KUKA KRL program: MyProgram_184().src

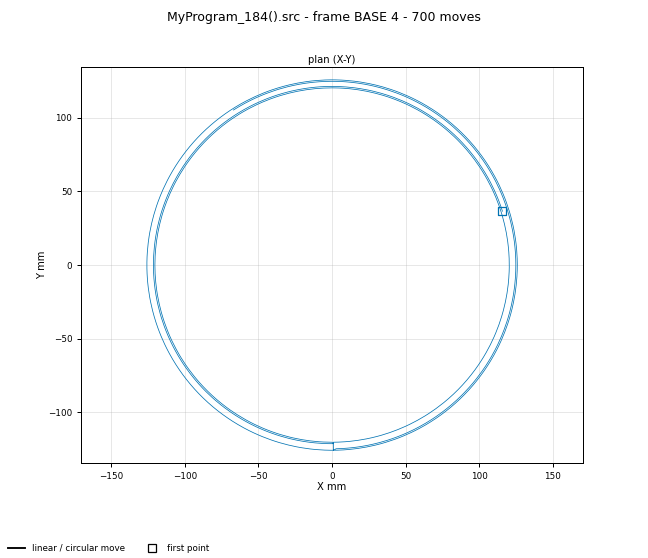
[picture p0: tool path of MyProgram_184().src in frame BASE 4, 700 of 700 moves have a stored position in this frame; points joined in program order, loops and branches not executed]
&ACCESS RVP
&REL 1
&PARAM TEMPLATE = C:\KRC\Roboter\Template\vorgabe
&PARAM EDITMASK = *
DEF MyProgram_184()
; ---- Setting reference (Base) ----
$BASE = BASE_DATA[4]

; --------------------------
; ---- Setting tool (TCP) ----
$TOOL = TOOL_DATA[3]
; --------------------------

$VEL.CP = VEL_APROX_PRINT
Startdeposition()
$VEL.CP = VEL_PRINT
LIN {X 115.7035,Y 36.5639,Z 134,A 13.9584,B 24.9464,C -1.6919,E1 25.152,E2 432.1213} C_DIS
LIN {X 114.6325,Y 39.7928,Z 134,A 15.5805,B 24.946,C -1.6976,E1 25.1505,E2 430.4949} C_DIS
LIN {X 113.3894,Y 43.2135,Z 134,A 17.3486,B 24.9455,C -1.7052,E1 25.1488,E2 428.7188} C_DIS
LIN {X 111.8645,Y 47.0156,Z 134,A 19.1684,B 24.9455,C -1.7052,E1 25.1469,E2 426.909} C_DIS
LIN {X 110.1148,Y 50.9782,Z 134,A 22.0831,B 24.9423,C -1.7548,E1 25.1434,E2 423.8932} C_DIS
LIN {X 107.5001,Y 56.2833,Z 134,A 23.673,B 24.9457,C -1.7024,E1 25.1415,E2 422.4351} C_DIS
LIN {X 105.7719,Y 59.4711,Z 134,A 25.7493,B 24.9442,C -1.7252,E1 25.1387,E2 420.3159} C_DIS
LIN {X 103.9941,Y 62.5285,Z 134,A 27.4667,B 24.9438,C -1.7321,E1 25.1362,E2 418.5912} C_DIS
LIN {X 101.7057,Y 66.1851,Z 134,A 30.2427,B 24.941,C -1.7744,E1 25.1319,E2 415.7292} C_DIS
LIN {X 98.373,Y 71.0443,Z 134,A 32.0344,B 24.9438,C -1.7322,E1 25.1292,E2 414.0459} C_DIS
LIN {X 96.2814,Y 73.854,Z 134,A 33.8484,B 24.943,C -1.7442,E1 25.1261,E2 412.2122} C_DIS
LIN {X 93.5282,Y 77.311,Z 134,A 35.9383,B 24.9426,C -1.7494,E1 25.1224,E2 410.1198} C_DIS
LIN {X 91.0407,Y 80.2255,Z 134,A 37.6345,B 24.9427,C -1.748,E1 25.1193,E2 408.4343} C_DIS
LIN {X 88.4927,Y 83.028,Z 134,A 39.4915,B 24.9422,C -1.7555,E1 25.1157,E2 406.568} C_DIS
LIN {X 86.0476,Y 85.5588,Z 134,A 41.1558,B 24.942,C -1.7592,E1 25.1125,E2 404.9019} C_DIS
LIN {X 82.9492,Y 88.5666,Z 134,A 43.0973,B 24.942,C -1.7588,E1 25.1086,E2 402.9694} C_DIS
LIN {X 80.4891,Y 90.8076,Z 134,A 44.7795,B 24.9415,C -1.7674,E1 25.1051,E2 401.2736} C_DIS
LIN {X 77.0787,Y 93.7202,Z 134,A 46.7789,B 24.9415,C -1.7658,E1 25.1008,E2 399.2857} C_DIS
LIN {X 73.9909,Y 96.1767,Z 134,A 48.7646,B 24.9409,C -1.7752,E1 25.0964,E2 397.2851} C_DIS
LIN {X 70.2941,Y 98.9108,Z 134,A 50.8899,B 24.9409,C -1.7768,E1 25.0916,E2 395.1636} C_DIS
LIN {X 65.6768,Y 102.035,Z 134,A 53.1943,B 24.9416,C -1.7653,E1 25.0864,E2 392.894} C_DIS
LIN {X 60.798,Y 105.0148,Z 134,A 56.0562,B 24.9408,C -1.7772,E1 25.0795,E2 390.0129} C_DIS
LIN {X 57.6858,Y 106.7564,Z 134,A 57.8367,B 24.9403,C -1.7842,E1 25.0751,E2 388.221} C_DIS
LIN {X 54.4905,Y 108.4215,Z 134,A 59.4404,B 24.9405,C -1.7818,E1 25.0711,E2 386.6275} C_DIS
LIN {X 52.1195,Y 109.5794,Z 134,A 61.0144,B 24.9393,C -1.7991,E1 25.0671,E2 385.0168} C_DIS
LIN {X 47.8558,Y 111.5078,Z 134,A 62.9444,B 24.9401,C -1.7882,E1 25.0622,E2 383.1172} C_DIS
LIN {X 41.891,Y 113.8847,Z 134,A 65.9124,B 24.9401,C -1.7882,E1 25.0545,E2 380.1559} C_DIS
LIN {X 37.7378,Y 115.3271,Z 134,A 68.2029,B 24.9393,C -1.8001,E1 25.0484,E2 377.8415} C_DIS
LIN {X 33.3869,Y 116.6617,Z 134,A 70.1325,B 24.9399,C -1.7913,E1 25.0433,E2 375.936} C_DIS
LIN {X 30.1024,Y 117.5501,Z 134,A 71.634,B 24.9401,C -1.7874,E1 25.0393,E2 374.4461} C_DIS
LIN {X 27.9003,Y 118.0931,Z 134,A 72.7821,B 24.9398,C -1.7917,E1 25.0361,E2 373.2896} C_DIS
LIN {X 24.6816,Y 118.8073,Z 134,A 74.2624,B 24.94,C -1.7889,E1 25.0321,E2 371.8179} C_DIS
LIN {X 21.5993,Y 119.4054,Z 134,A 75.6288,B 24.9403,C -1.7841,E1 25.0284,E2 370.4644} C_DIS
LIN {X 19.0604,Y 119.8377,Z 134,A 77.1116,B 24.9395,C -1.7969,E1 25.0242,E2 368.9527} C_DIS
LIN {X 15.3542,Y 120.3684,Z 134,A 79.0415,B 24.9389,C -1.8049,E1 25.0188,E2 367.0054} C_DIS
LIN {X 9.5046,Y 120.9722,Z 134,A 81.5766,B 24.9397,C -1.7939,E1 25.0119,E2 364.4979} C_DIS
LIN {X 4.175,Y 121.2715,Z 134,A 84.0832,B 24.9397,C -1.7932,E1 25.0049,E2 361.9938} C_DIS
LIN {X -3.3352,Y 121.2974,Z 134,A 87.3752,B 24.9406,C -1.7807,E1 24.9958,E2 358.7316} C_DIS
LIN {X -8.0647,Y 121.0756,Z 134,A 89.9951,B 24.9394,C -1.7975,E1 24.9884,E2 356.0711} C_DIS
LIN {X -10.9283,Y 120.8515,Z 134,A 91.8989,B 24.9378,C -1.8221,E1 24.9829,E2 354.1081} C_DIS
LIN {X -15.3011,Y 120.3754,Z 134,A 93.3926,B 24.9397,C -1.794,E1 24.9789,E2 352.68} C_DIS
LIN {X -18.4282,Y 119.9356,Z 134,A 94.8364,B 24.9399,C -1.7909,E1 24.975,E2 351.2425} C_DIS
LIN {X -23.1856,Y 119.108,Z 134,A 97.1985,B 24.9398,C -1.7928,E1 24.9685,E2 348.8734} C_DIS
LIN {X -27.8258,Y 118.1111,Z 134,A 99.3651,B 24.9401,C -1.7874,E1 24.9626,E2 346.7169} C_DIS
LIN {X -30.2861,Y 117.5034,Z 134,A 100.7404,B 24.9397,C -1.7943,E1 24.9588,E2 345.3231} C_DIS
LIN {X -33.7688,Y 116.5499,Z 134,A 102.3978,B 24.9399,C -1.7903,E1 24.9544,E2 343.6725} C_DIS
LIN {X -36.9708,Y 115.5736,Z 134,A 103.902,B 24.9403,C -1.785,E1 24.9504,E2 342.1783} C_DIS
LIN {X -40.2534,Y 114.4728,Z 134,A 105.5084,B 24.9405,C -1.7817,E1 24.9462,E2 340.5768} C_DIS
LIN {X -44.5725,Y 112.8618,Z 134,A 107.6515,B 24.9408,C -1.7772,E1 24.9406,E2 338.4398} C_DIS
LIN {X -47.2777,Y 111.7551,Z 134,A 109.0429,B 24.9408,C -1.7758,E1 24.937,E2 337.0487} C_DIS
LIN {X -49.6424,Y 110.7236,Z 134,A 110.3052,B 24.9408,C -1.7759,E1 24.9338,E2 335.783} C_DIS
LIN {X -52.8834,Y 109.2145,Z 134,A 111.9711,B 24.9411,C -1.7722,E1 24.9296,E2 334.1216} C_DIS
LIN {X -55.7632,Y 107.7732,Z 134,A 113.7041,B 24.9407,C -1.7792,E1 24.9252,E2 332.3674} C_DIS
LIN {X -59.7868,Y 105.5944,Z 134,A 115.8609,B 24.9409,C -1.7752,E1 24.9199,E2 330.2138} C_DIS
LIN {X -63.7405,Y 103.2558,Z 134,A 117.8702,B 24.9417,C -1.7641,E1 24.9152,E2 328.2248} C_DIS
LIN {X -66.727,Y 101.3509,Z 134,A 119.6469,B 24.9416,C -1.7655,E1 24.911,E2 326.4391} C_DIS
LIN {X -70.2515,Y 98.9412,Z 134,A 121.7402,B 24.9416,C -1.7648,E1 24.9062,E2 324.3403} C_DIS
LIN {X -73.8247,Y 96.3038,Z 134,A 123.7505,B 24.9422,C -1.7565,E1 24.9017,E2 322.3425} C_DIS
LIN {X -76.7002,Y 94.0297,Z 134,A 125.5201,B 24.9423,C -1.7544,E1 24.8979,E2 320.5713} C_DIS
LIN {X -79.9876,Y 91.25,Z 134,A 127.6022,B 24.9425,C -1.7519,E1 24.8935,E2 318.487} C_DIS
LIN {X -83.0686,Y 88.4544,Z 134,A 129.5856,B 24.9427,C -1.7481,E1 24.8894,E2 316.5046} C_DIS
LIN {X -85.974,Y 85.6329,Z 134,A 131.4349,B 24.9432,C -1.7407,E1 24.8858,E2 314.6652} C_DIS
LIN {X -88.6608,Y 82.8481,Z 134,A 133.3372,B 24.9433,C -1.7394,E1 24.8821,E2 312.7578} C_DIS
LIN {X -91.6123,Y 79.5724,Z 134,A 135.3816,B 24.9438,C -1.7323,E1 24.8783,E2 310.7208} C_DIS
LIN {X -94.2611,Y 76.4161,Z 134,A 137.3068,B 24.9442,C -1.7263,E1 24.8749,E2 308.8012} C_DIS
LIN {X -96.6023,Y 73.4344,Z 134,A 139.2073,B 24.9442,C -1.7263,E1 24.8716,E2 306.8918} C_DIS
LIN {X -99.1829,Y 69.9088,Z 134,A 141.2347,B 24.9446,C -1.719,E1 24.8684,E2 304.8718} C_DIS
LIN {X -101.1758,Y 66.993,Z 134,A 143.5278,B 24.9432,C -1.7416,E1 24.8647,E2 302.5132} C_DIS
LIN {X -103.799,Y 62.8512,Z 134,A 144.9179,B 24.9462,C -1.6946,E1 24.8629,E2 301.2282} C_DIS
LIN {X -105.1935,Y 60.4893,Z 134,A 147.3202,B 24.9433,C -1.7391,E1 24.8594,E2 298.7073} C_DIS
LIN {X -107.8811,Y 55.552,Z 134,A 149.3952,B 24.9455,C -1.7057,E1 24.8568,E2 296.7007} C_DIS
LIN {X -110.2068,Y 50.7793,Z 134,A 151.6913,B 24.9465,C -1.6889,E1 24.854,E2 294.4321} C_DIS
LIN {X -111.6204,Y 47.5954,Z 134,A 153.4183,B 24.9466,C -1.6874,E1 24.8521,E2 292.6993} C_DIS
LIN {X -113.0711,Y 44.0342,Z 134,A 155.1365,B 24.9473,C -1.6776,E1 24.8503,E2 290.9949} C_DIS
LIN {X -114.1922,Y 41.0394,Z 134,A 156.6516,B 24.9475,C -1.673,E1 24.8489,E2 289.482} C_DIS
LIN {X -115.5432,Y 37.0659,Z 134,A 158.3702,B 24.9486,C -1.6554,E1 24.8474,E2 287.7957} C_DIS
LIN {X -116.4116,Y 34.241,Z 134,A 160.0742,B 24.9481,C -1.6642,E1 24.846,E2 286.0608} C_DIS
LIN {X -117.2688,Y 31.1789,Z 134,A 161.5904,B 24.9484,C -1.6601,E1 24.8449,E2 284.5457} C_DIS
LIN {X -118.2375,Y 27.2779,Z 134,A 163.5201,B 24.9487,C -1.6553,E1 24.8436,E2 282.6161} C_DIS
LIN {X -119.0118,Y 23.6769,Z 134,A 165.3867,B 24.9487,C -1.6551,E1 24.8426,E2 280.7389} C_DIS
LIN {X -119.8062,Y 19.2641,Z 134,A 167.3156,B 24.9496,C -1.6401,E1 24.8417,E2 278.8344} C_DIS
LIN {X -120.2979,Y 15.8923,Z 134,A 169.0647,B 24.9496,C -1.6409,E1 24.841,E2 277.0729} C_DIS
LIN {X -120.6915,Y 12.5658,Z 134,A 170.5144,B 24.9502,C -1.63,E1 24.8406,E2 275.6404} C_DIS
LIN {X -120.9954,Y 9.1867,Z 134,A 171.9906,B 24.9509,C -1.6193,E1 24.8402,E2 274.1809} C_DIS
LIN {X -121.1631,Y 6.6297,Z 134,A 173.4769,B 24.9504,C -1.6273,E1 24.84,E2 272.6667} C_DIS
LIN {X -121.3239,Y 2.1708,Z 134,A 175.2986,B 24.9515,C -1.6081,E1 24.8398,E2 270.8797} C_DIS
LIN {X -121.3431,Y -0.5711,Z 134,A 176.9721,B 24.9508,C -1.6202,E1 24.8398,E2 269.1673} C_DIS
LIN {X -121.2455,Y -4.8701,Z 134,A 178.9278,B 24.9514,C -1.6103,E1 24.84,E2 267.2233} C_DIS
LIN {X -121.0159,Y -8.9065,Z 134,A -179.1471,B 24.9517,C -1.6048,E1 24.8403,E2 265.2998} C_DIS
LIN {X -120.6571,Y -12.8846,Z 134,A -177.3052,B 24.9522,C -1.5968,E1 24.8408,E2 263.466} C_DIS
LIN {X -120.1951,Y -16.6592,Z 134,A -175.6228,B 24.9529,C -1.5861,E1 24.8414,E2 261.799} C_DIS
LIN {X -119.6956,Y -19.927,Z 134,A -173.8537,B 24.9526,C -1.5901,E1 24.8422,E2 260.0098} C_DIS
LIN {X -118.9436,Y -24.0119,Z 134,A -172.2153,B 24.9538,C -1.5699,E1 24.843,E2 258.4099} C_DIS
LIN {X -118.3366,Y -26.844,Z 134,A -170.5132,B 24.9532,C -1.5801,E1 24.8441,E2 256.6735} C_DIS
LIN {X -117.4748,Y -30.3988,Z 134,A -168.8828,B 24.9538,C -1.5705,E1 24.8452,E2 255.0565} C_DIS
LIN {X -116.8617,Y -32.6716,Z 134,A -167.7228,B 24.9538,C -1.5692,E1 24.846,E2 253.8929} C_DIS
LIN {X -115.937,Y -35.8163,Z 134,A -166.0643,B 24.9538,C -1.5692,E1 24.8474,E2 252.2247} C_DIS
LIN {X -114.0898,Y -41.3233,Z 134,A -163.3944,B 24.9545,C -1.5578,E1 24.8498,E2 249.567} C_DIS
LIN {X -112.8337,Y -44.6447,Z 134,A -161.6144,B 24.9545,C -1.5573,E1 24.8516,E2 247.7781} C_DIS
LIN {X -111.3837,Y -48.1428,Z 134,A -159.8769,B 24.955,C -1.5498,E1 24.8535,E2 246.0487} C_DIS
LIN {X -109.6161,Y -52.0427,Z 134,A -157.8435,B 24.9553,C -1.5445,E1 24.8559,E2 244.0169} C_DIS
LIN {X -108.1159,Y -55.0909,Z 134,A -156.2403,B 24.9556,C -1.54,E1 24.8579,E2 242.4159} C_DIS
LIN {X -106.6023,Y -57.9696,Z 134,A -154.5061,B 24.9553,C -1.5444,E1 24.8602,E2 240.662} C_DIS
LIN {X -104.9695,Y -60.8761,Z 134,A -153.0536,B 24.9559,C -1.5347,E1 24.8622,E2 239.225} C_DIS
LIN {X -102.9788,Y -64.1863,Z 134,A -151.2733,B 24.9563,C -1.5279,E1 24.8648,E2 237.4517} C_DIS
LIN {X -101.0347,Y -67.2051,Z 134,A -149.67,B 24.9567,C -1.5194,E1 24.8672,E2 235.8607} C_DIS
LIN {X -99.0903,Y -70.0402,Z 134,A -147.8584,B 24.9565,C -1.5236,E1 24.8701,E2 234.0301} C_DIS
LIN {X -96.1694,Y -74.0005,Z 134,A -145.1153,B 24.9558,C -1.5365,E1 24.8748,E2 231.2432} C_DIS
LIN {X -93.6787,Y -77.1291,Z 134,A -143.9263,B 24.9578,C -1.5008,E1 24.8768,E2 230.1336} C_DIS
LIN {X -90.6682,Y -80.6469,Z 134,A -141.4937,B 24.9575,C -1.5067,E1 24.8813,E2 227.6761} C_DIS
LIN {X -88.0575,Y -83.4893,Z 134,A -139.7866,B 24.958,C -1.4974,E1 24.8845,E2 225.9834} C_DIS
LIN {X -85.706,Y -85.901,Z 134,A -137.2019,B 24.9556,C -1.5388,E1 24.8898,E2 223.2894} C_DIS
LIN {X -81.4811,Y -89.9185,Z 134,A -135.4738,B 24.9586,C -1.4868,E1 24.8931,E2 221.6779} C_DIS
LIN {X -79.3216,Y -91.8292,Z 134,A -133.8806,B 24.9582,C -1.4945,E1 24.8965,E2 220.0602} C_DIS
LIN {X -75.4367,Y -95.0464,Z 134,A -131.6679,B 24.9588,C -1.4824,E1 24.9013,E2 217.868} C_DIS
LIN {X -72.7704,Y -97.1036,Z 134,A -129.8745,B 24.9585,C -1.4887,E1 24.9053,E2 216.0531} C_DIS
LIN {X -68.7433,Y -99.9943,Z 134,A -127.561,B 24.9588,C -1.4835,E1 24.9106,E2 213.7441} C_DIS
LIN {X -65.3047,Y -102.2732,Z 134,A -125.5443,B 24.9588,C -1.4835,E1 24.9153,E2 211.7207} C_DIS
LIN {X -61.2708,Y -104.7399,Z 134,A -123.3979,B 24.9592,C -1.4762,E1 24.9204,E2 209.5851} C_DIS
LIN {X -57.7406,Y -106.7269,Z 134,A -121.3991,B 24.9592,C -1.4775,E1 24.9253,E2 207.5775} C_DIS
LIN {X -54.9349,Y -108.1953,Z 134,A -119.7449,B 24.9588,C -1.4829,E1 24.9295,E2 205.906} C_DIS
LIN {X -51.7077,Y -109.7762,Z 134,A -118.1742,B 24.9592,C -1.475,E1 24.9334,E2 204.35} C_DIS
LIN {X -48.0474,Y -111.4249,Z 134,A -116.0306,B 24.9587,C -1.4844,E1 24.939,E2 202.1791} C_DIS
LIN {X -44.7756,Y -112.7813,Z 134,A -114.7859,B 24.9599,C -1.4629,E1 24.9421,E2 200.9825} C_DIS
LIN {X -41.9536,Y -113.8613,Z 134,A -113.1664,B 24.9595,C -1.4705,E1 24.9464,E2 199.3418} C_DIS
LIN {X -38.1159,Y -115.2012,Z 134,A -111.3665,B 24.9599,C -1.4634,E1 24.9511,E2 197.5553} C_DIS
LIN {X -35.1633,Y -116.1368,Z 134,A -109.8351,B 24.9598,C -1.4655,E1 24.9552,E2 196.0163} C_DIS
LIN {X -31.9316,Y -117.0681,Z 134,A -108.3835,B 24.9602,C -1.4581,E1 24.9591,E2 194.58} C_DIS
LIN {X -29.7459,Y -117.6405,Z 134,A -107.3059,B 24.9602,C -1.458,E1 24.962,E2 193.5011} C_DIS
LIN {X -26.6223,Y -118.3872,Z 134,A -105.6103,B 24.9598,C -1.4656,E1 24.9666,E2 191.7853} C_DIS
LIN {X -23.1435,Y -119.1161,Z 134,A -103.9475,B 24.9598,C -1.4641,E1 24.9712,E2 190.124} C_DIS
LIN {X -19.3211,Y -119.7967,Z 134,A -102.0752,B 24.9598,C -1.4654,E1 24.9764,E2 188.247} C_DIS
LIN {X -15.4126,Y -120.3608,Z 134,A -100.1288,B 24.9596,C -1.4688,E1 24.9818,E2 186.2908} C_DIS
LIN {X -11.4809,Y -120.7988,Z 134,A -97.738,B 24.9582,C -1.4935,E1 24.9886,E2 183.8403} C_DIS
LIN {X -6.2901,Y -121.1802,Z 134,A -95.9521,B 24.96,C -1.4616,E1 24.9934,E2 182.1294} C_DIS
LIN {X -2.8879,Y -121.3098,Z 134,A -94.4302,B 24.9602,C -1.4578,E1 24.9976,E2 180.6164} C_DIS
LIN {X 0.8558,Y -121.3391,Z 134,A -92.6939,B 24.9602,C -1.4567,E1 25.0024,E2 178.8827} C_DIS
Enddeposition()
LIN {X 0.8558,Y -121.3391,Z 134,A -92.6939,B 24.9602,C -1.4567,E1 25.0024,E2 178.8827} C_DIS
Startdeposition()
$VEL.CP = VEL_PRINT
LIN {X -0.059,Y -120.3485,Z 134,A -93.8009,B 24.961,C -1.4425,E1 24.9993,E2 180.0232} C_DIS
LIN {X -3.0062,Y -120.3099,Z 134,A -95.2081,B 24.961,C -1.4421,E1 24.9953,E2 181.4315} C_DIS
LIN {X -5.9627,Y -120.1991,Z 134,A -96.6041,B 24.961,C -1.4426,E1 24.9914,E2 182.8267} C_DIS
LIN {X -8.8785,Y -120.019,Z 134,A -97.9907,B 24.961,C -1.4428,E1 24.9876,E2 184.2134} C_DIS
LIN {X -12.3601,Y -119.7115,Z 134,A -99.5673,B 24.9608,C -1.4469,E1 24.9832,E2 185.7811} C_DIS
LIN {X -14.8176,Y -119.4325,Z 134,A -100.8252,B 24.961,C -1.4434,E1 24.9797,E2 187.0481} C_DIS
LIN {X -17.684,Y -119.0423,Z 134,A -102.2326,B 24.961,C -1.4423,E1 24.9758,E2 188.4592} C_DIS
LIN {X -20.6314,Y -118.5665,Z 134,A -103.7084,B 24.9611,C -1.4403,E1 24.9717,E2 189.9412} C_DIS
LIN {X -23.5237,Y -118.0262,Z 134,A -105.054,B 24.961,C -1.4433,E1 24.968,E2 191.281} C_DIS
LIN {X -26.4266,Y -117.41,Z 134,A -106.4445,B 24.9609,C -1.445,E1 24.9642,E2 192.6692} C_DIS
LIN {X -29.2945,Y -116.7272,Z 134,A -107.8634,B 24.9609,C -1.4451,E1 24.9604,E2 194.0899} C_DIS
LIN {X -32.331,Y -115.9224,Z 134,A -109.2925,B 24.9607,C -1.4491,E1 24.9566,E2 195.5118} C_DIS
LIN {X -34.9345,Y -115.1649,Z 134,A -110.6655,B 24.9608,C -1.4463,E1 24.9529,E2 196.8937} C_DIS
LIN {X -37.7894,Y -114.2598,Z 134,A -112.0693,B 24.9608,C -1.4484,E1 24.9491,E2 198.295} C_DIS
LIN {X -41.217,Y -113.0691,Z 134,A -113.9242,B 24.9609,C -1.4442,E1 24.9442,E2 200.1637} C_DIS
LIN {X -44.7088,Y -111.734,Z 134,A -115.696,B 24.9609,C -1.4463,E1 24.9396,E2 201.9343} C_DIS
LIN {X -47.4697,Y -110.5893,Z 134,A -117.0016,B 24.9604,C -1.4531,E1 24.9363,E2 203.2268} C_DIS
LIN {X -50.4526,Y -109.2602,Z 134,A -118.4573,B 24.9601,C -1.4593,E1 24.9326,E2 204.6712} C_DIS
LIN {X -52.8382,Y -108.1276,Z 134,A -119.8337,B 24.9603,C -1.4554,E1 24.9291,E2 206.0602} C_DIS
LIN {X -55.4725,Y -106.8005,Z 134,A -121.2038,B 24.9601,C -1.4588,E1 24.9257,E2 207.4262} C_DIS
LIN {X -58.7025,Y -105.061,Z 134,A -123.1582,B 24.9605,C -1.4519,E1 24.9209,E2 209.4024} C_DIS
LIN {X -62.1921,Y -103.0333,Z 134,A -124.8451,B 24.9598,C -1.4651,E1 24.9169,E2 211.0629} C_DIS
LIN {X -64.3939,Y -101.6718,Z 134,A -126.1656,B 24.9598,C -1.4631,E1 24.9137,E2 212.3925} C_DIS
LIN {X -66.8616,Y -100.0661,Z 134,A -127.5697,B 24.9598,C -1.4653,E1 24.9105,E2 213.796} C_DIS
LIN {X -69.3066,Y -98.3885,Z 134,A -128.9842,B 24.9597,C -1.4675,E1 24.9072,E2 215.2099} C_DIS
LIN {X -71.6968,Y -96.6608,Z 134,A -130.5546,B 24.9599,C -1.4627,E1 24.9036,E2 216.7975} C_DIS
LIN {X -75.2403,Y -93.9295,Z 134,A -132.6933,B 24.9597,C -1.4662,E1 24.8989,E2 218.9356} C_DIS
LIN {X -78.6292,Y -91.1107,Z 134,A -134.8021,B 24.9595,C -1.4699,E1 24.8945,E2 221.0439} C_DIS
LIN {X -81.5322,Y -88.5224,Z 134,A -136.6341,B 24.9593,C -1.4745,E1 24.8907,E2 222.8723} C_DIS
LIN {X -84.611,Y -85.5849,Z 134,A -138.6871,B 24.9591,C -1.4776,E1 24.8866,E2 224.9264} C_DIS
LIN {X -87.6778,Y -82.4399,Z 134,A -140.8004,B 24.9589,C -1.4813,E1 24.8825,E2 227.0402} C_DIS
LIN {X -90.6478,Y -79.1623,Z 134,A -142.9165,B 24.9587,C -1.4856,E1 24.8785,E2 229.1553} C_DIS
LIN {X -93.5153,Y -75.7539,Z 134,A -145.0332,B 24.9584,C -1.4909,E1 24.8748,E2 231.2694} C_DIS
LIN {X -95.9907,Y -72.5913,Z 134,A -146.7317,B 24.9576,C -1.5048,E1 24.8719,E2 232.9427} C_DIS
LIN {X -97.565,Y -70.4614,Z 134,A -148.1999,B 24.9579,C -1.499,E1 24.8695,E2 234.4319} C_DIS
LIN {X -99.5103,Y -67.6866,Z 134,A -149.6224,B 24.9572,C -1.5114,E1 24.8673,E2 235.832} C_DIS
LIN {X -101.1748,Y -65.1727,Z 134,A -151.0459,B 24.957,C -1.5156,E1 24.8651,E2 237.2525} C_DIS
LIN {X -102.4843,Y -63.0928,Z 134,A -152.3,B 24.957,C -1.5151,E1 24.8632,E2 238.5141} C_DIS
LIN {X -103.9976,Y -60.5664,Z 134,A -153.7836,B 24.957,C -1.5154,E1 24.8611,E2 240.0047} C_DIS
LIN {X -105.8233,Y -57.3172,Z 134,A -155.6806,B 24.957,C -1.5151,E1 24.8585,E2 241.9126} C_DIS
LIN {X -107.7105,Y -53.6837,Z 134,A -157.5254,B 24.9564,C -1.525,E1 24.8562,E2 243.7434} C_DIS
LIN {X -108.8191,Y -51.3999,Z 134,A -158.6958,B 24.9561,C -1.5301,E1 24.8548,E2 244.9081} C_DIS
LIN {X -110.2728,Y -48.2018,Z 134,A -160.5624,B 24.9563,C -1.5267,E1 24.8527,E2 246.793} C_DIS
LIN {X -111.7587,Y -44.6476,Z 134,A -162.2158,B 24.9556,C -1.5398,E1 24.8509,E2 248.4245} C_DIS
LIN {X -112.8025,Y -41.9399,Z 134,A -163.616,B 24.9554,C -1.5431,E1 24.8495,E2 249.8247} C_DIS
LIN {X -113.7954,Y -39.1658,Z 134,A -165.0244,B 24.9552,C -1.5471,E1 24.8482,E2 251.2315} C_DIS
LIN {X -114.7409,Y -36.3033,Z 134,A -166.5723,B 24.9552,C -1.5467,E1 24.8469,E2 252.7893} C_DIS
LIN {X -115.989,Y -32.0931,Z 134,A -168.5687,B 24.9546,C -1.5572,E1 24.8454,E2 254.7724} C_DIS
LIN {X -116.8742,Y -28.7052,Z 134,A -170.1543,B 24.9541,C -1.5658,E1 24.8443,E2 256.3466} C_DIS
LIN {X -117.4229,Y -26.3699,Z 134,A -171.5551,B 24.9545,C -1.5584,E1 24.8434,E2 257.7732} C_DIS
LIN {X -118.0377,Y -23.4676,Z 134,A -172.8126,B 24.9538,C -1.5694,E1 24.8427,E2 259.0118} C_DIS
LIN {X -118.5777,Y -20.5689,Z 134,A -174.2393,B 24.9536,C -1.5729,E1 24.842,E2 260.4388} C_DIS
LIN {X -119.0459,Y -17.6584,Z 134,A -175.6605,B 24.9534,C -1.5767,E1 24.8414,E2 261.8594} C_DIS
LIN {X -119.4572,Y -14.6105,Z 134,A -177.0973,B 24.9531,C -1.5825,E1 24.8409,E2 263.2909} C_DIS
LIN {X -119.7732,Y -11.7382,Z 134,A -178.5121,B 24.9529,C -1.5854,E1 24.8405,E2 264.7075} C_DIS
LIN {X -120.0246,Y -8.8018,Z 134,A -179.9595,B 24.9527,C -1.588,E1 24.8401,E2 266.1571} C_DIS
LIN {X -120.202,Y -5.9048,Z 134,A 178.6956,B 24.9524,C -1.5941,E1 24.8399,E2 267.4957} C_DIS
LIN {X -120.3148,Y -2.8264,Z 134,A 177.2361,B 24.9521,C -1.5992,E1 24.8399,E2 268.9519} C_DIS
LIN {X -120.3498,Y 0.0029,Z 134,A 175.7959,B 24.9521,C -1.5996,E1 24.8398,E2 270.3997} C_DIS
LIN {X -120.3097,Y 3.0112,Z 134,A 174.402,B 24.9517,C -1.606,E1 24.8398,E2 271.7869} C_DIS
LIN {X -120.1955,Y 6.0351,Z 134,A 172.874,B 24.9517,C -1.607,E1 24.8401,E2 273.3216} C_DIS
LIN {X -119.9021,Y 10.3386,Z 134,A 170.8937,B 24.951,C -1.6168,E1 24.8405,E2 275.2903} C_DIS
LIN {X -119.6132,Y 13.2739,Z 134,A 169.4859,B 24.9507,C -1.6213,E1 24.8409,E2 276.6961} C_DIS
LIN {X -119.2467,Y 16.2466,Z 134,A 167.9115,B 24.9508,C -1.6197,E1 24.8414,E2 278.2836} C_DIS
LIN {X -118.8131,Y 19.1629,Z 134,A 166.6178,B 24.9503,C -1.6289,E1 24.842,E2 279.563} C_DIS
LIN {X -118.3073,Y 22.068,Z 134,A 165.2074,B 24.95,C -1.6332,E1 24.8427,E2 280.9716} C_DIS
LIN {X -117.728,Y 24.9723,Z 134,A 163.7902,B 24.9498,C -1.6375,E1 24.8435,E2 282.3869} C_DIS
LIN {X -117.0609,Y 27.9311,Z 134,A 162.2615,B 24.9497,C -1.6386,E1 24.8445,E2 283.922} C_DIS
LIN {X -116.3607,Y 30.7177,Z 134,A 160.9611,B 24.9492,C -1.6458,E1 24.8454,E2 285.2127} C_DIS
LIN {X -115.5852,Y 33.518,Z 134,A 159.5689,B 24.949,C -1.6499,E1 24.8464,E2 286.6033} C_DIS
LIN {X -114.7144,Y 36.3861,Z 134,A 158.134,B 24.9487,C -1.6541,E1 24.8476,E2 288.0364} C_DIS
LIN {X -113.5174,Y 39.9678,Z 134,A 156.1495,B 24.9489,C -1.6519,E1 24.8494,E2 290.0374} C_DIS
LIN {X -112.2781,Y 43.3244,Z 134,A 154.6101,B 24.9481,C -1.6642,E1 24.8509,E2 291.5562} C_DIS
LIN {X -111.165,Y 46.1053,Z 134,A 153.1751,B 24.9479,C -1.6682,E1 24.8524,E2 292.9896} C_DIS
LIN {X -110.0203,Y 48.7744,Z 134,A 151.7849,B 24.9476,C -1.6721,E1 24.854,E2 294.3781} C_DIS
LIN {X -108.5073,Y 52.0525,Z 134,A 150.1963,B 24.9469,C -1.6829,E1 24.8558,E2 295.9497} C_DIS
LIN {X -107.4529,Y 54.1972,Z 134,A 148.9155,B 24.9471,C -1.6803,E1 24.8574,E2 297.2436} C_DIS
LIN {X -106.1219,Y 56.7617,Z 134,A 147.5276,B 24.9469,C -1.6838,E1 24.8592,E2 298.6304} C_DIS
LIN {X -104.4224,Y 59.8307,Z 134,A 145.9744,B 24.9462,C -1.6937,E1 24.8613,E2 300.1682} C_DIS
LIN {X -103.2281,Y 61.8688,Z 134,A 144.6987,B 24.9464,C -1.6906,E1 24.8632,E2 301.4579} C_DIS
LIN {X -101.6877,Y 64.3688,Z 134,A 143.2941,B 24.9462,C -1.6943,E1 24.8652,E2 302.8608} C_DIS
LIN {X -100.0621,Y 66.8676,Z 134,A 141.8738,B 24.9459,C -1.6983,E1 24.8674,E2 304.2787} C_DIS
LIN {X -98.3935,Y 69.2995,Z 134,A 140.3062,B 24.9461,C -1.6953,E1 24.87,E2 305.8612} C_DIS
LIN {X -95.7997,Y 72.8439,Z 134,A 138.1864,B 24.9459,C -1.6998,E1 24.8735,E2 307.9805} C_DIS
LIN {X -93.0286,Y 76.3508,Z 134,A 136.0498,B 24.9455,C -1.7052,E1 24.8772,E2 310.1143} C_DIS
LIN {X -90.1594,Y 79.7181,Z 134,A 133.9784,B 24.9451,C -1.7121,E1 24.881,E2 312.1785} C_DIS
LIN {X -87.3186,Y 82.8206,Z 134,A 132.0334,B 24.9446,C -1.7197,E1 24.8847,E2 314.1142} C_DIS
LIN {X -84.5583,Y 85.6372,Z 134,A 130.0316,B 24.9446,C -1.719,E1 24.8886,E2 316.1261} C_DIS
LIN {X -81.3523,Y 88.6877,Z 134,A 127.9416,B 24.9443,C -1.7247,E1 24.8929,E2 318.2109} C_DIS
LIN {X -78.0613,Y 91.5978,Z 134,A 125.8122,B 24.944,C -1.7279,E1 24.8974,E2 320.3411} C_DIS
LIN {X -74.6059,Y 94.4339,Z 134,A 123.6763,B 24.9438,C -1.7322,E1 24.902,E2 322.4747} C_DIS
LIN {X -71.0502,Y 97.1372,Z 134,A 121.5641,B 24.9434,C -1.7374,E1 24.9067,E2 324.5823} C_DIS
LIN {X -68.0404,Y 99.2683,Z 134,A 119.94,B 24.9428,C -1.7466,E1 24.9104,E2 326.1899} C_DIS
LIN {X -65.5877,Y 100.9057,Z 134,A 118.5445,B 24.9426,C -1.7497,E1 24.9137,E2 327.5825} C_DIS
LIN {X -63.0956,Y 102.4826,Z 134,A 117.1388,B 24.9424,C -1.7523,E1 24.917,E2 328.9865} C_DIS
LIN {X -60.5664,Y 103.9977,Z 134,A 115.5605,B 24.9428,C -1.7473,E1 24.9208,E2 330.5815} C_DIS
LIN {X -56.7119,Y 106.1487,Z 134,A 113.5796,B 24.9422,C -1.7562,E1 24.9256,E2 332.5469} C_DIS
LIN {X -54.0985,Y 107.5031,Z 134,A 112.1867,B 24.942,C -1.7589,E1 24.9291,E2 333.9371} C_DIS
LIN {X -51.4085,Y 108.815,Z 134,A 110.5932,B 24.9423,C -1.7539,E1 24.9332,E2 335.5467} C_DIS
LIN {X -47.4184,Y 110.6115,Z 134,A 108.6686,B 24.9417,C -1.7639,E1 24.938,E2 337.452} C_DIS
LIN {X -44.6529,Y 111.7565,Z 134,A 107.223,B 24.9417,C -1.765,E1 24.9418,E2 338.8981} C_DIS
LIN {X -41.9259,Y 112.8077,Z 134,A 105.8448,B 24.9414,C -1.7675,E1 24.9454,E2 340.2735} C_DIS
LIN {X -38.4066,Y 114.0543,Z 134,A 104.0782,B 24.9413,C -1.7702,E1 24.95,E2 342.037} C_DIS
LIN {X -34.88,Y 115.1816,Z 134,A 102.3087,B 24.9412,C -1.772,E1 24.9547,E2 343.8054} C_DIS
LIN {X -32.0922,Y 115.9892,Z 134,A 100.9125,B 24.9411,C -1.7728,E1 24.9585,E2 345.2018} C_DIS
LIN {X -29.1964,Y 116.7521,Z 134,A 99.3963,B 24.9413,C -1.7702,E1 24.9626,E2 346.7264} C_DIS
LIN {X -26.3583,Y 117.4256,Z 134,A 98.1022,B 24.9409,C -1.7757,E1 24.9661,E2 348.0091} C_DIS
LIN {X -23.4506,Y 118.0411,Z 134,A 96.6877,B 24.9409,C -1.7769,E1 24.97,E2 349.4224} C_DIS
LIN {X -20.5574,Y 118.5797,Z 134,A 95.1527,B 24.9411,C -1.772,E1 24.9742,E2 350.9706} C_DIS
LIN {X -17.6519,Y 119.0469,Z 134,A 93.8606,B 24.9408,C -1.7778,E1 24.9777,E2 352.25} C_DIS
LIN {X -14.1946,Y 119.5068,Z 134,A 92.2803,B 24.9405,C -1.7825,E1 24.9821,E2 353.8205} C_DIS
LIN {X -11.6118,Y 119.7854,Z 134,A 90.9807,B 24.9405,C -1.7803,E1 24.9857,E2 355.126} C_DIS
LIN {X -8.7486,Y 120.0285,Z 134,A 89.6082,B 24.9405,C -1.7807,E1 24.9895,E2 356.4981} C_DIS
LIN {X -5.8859,Y 120.203,Z 134,A 88.1201,B 24.9409,C -1.7757,E1 24.9937,E2 357.9985} C_DIS
LIN {X -2.8562,Y 120.314,Z 134,A 86.8161,B 24.9405,C -1.7824,E1 24.9973,E2 359.2868} C_DIS
LIN {X 0.0679,Y 120.3484,Z 134,A 85.2139,B 24.9411,C -1.7732,E1 25.0018,E2 360.9107} C_DIS
LIN {X 4.4953,Y 120.2631,Z 134,A 83.2962,B 24.9405,C -1.7821,E1 25.0071,E2 362.8071} C_DIS
LIN {X 7.6324,Y 120.1048,Z 134,A 81.7129,B 24.9407,C -1.7781,E1 25.0116,E2 364.3992} C_DIS
LIN {X 11.87,Y 119.7606,Z 134,A 79.7848,B 24.9405,C -1.7823,E1 25.0169,E2 366.3163} C_DIS
LIN {X 14.7962,Y 119.435,Z 134,A 78.3819,B 24.9405,C -1.782,E1 25.0208,E2 367.719} C_DIS
LIN {X 17.6682,Y 119.0445,Z 134,A 76.9788,B 24.9405,C -1.7805,E1 25.0247,E2 369.1243} C_DIS
LIN {X 20.6198,Y 118.5686,Z 134,A 75.5506,B 24.9406,C -1.7798,E1 25.0286,E2 370.5527} C_DIS
LIN {X 23.5374,Y 118.0234,Z 134,A 74.1495,B 24.9406,C -1.7798,E1 25.0325,E2 371.9522} C_DIS
LIN {X 26.421,Y 117.4112,Z 134,A 72.7642,B 24.9406,C -1.7798,E1 25.0362,E2 373.3353} C_DIS
LIN {X 29.2898,Y 116.7284,Z 134,A 71.3484,B 24.9407,C -1.7785,E1 25.0401,E2 374.7523} C_DIS
LIN {X 32.1415,Y 115.9755,Z 134,A 69.9596,B 24.9407,C -1.7783,E1 25.0438,E2 376.1394} C_DIS
LIN {X 34.9305,Y 115.1662,Z 134,A 68.5517,B 24.9409,C -1.7761,E1 25.0476,E2 377.5501} C_DIS
LIN {X 38.3389,Y 114.0768,Z 134,A 66.8297,B 24.941,C -1.7738,E1 25.0522,E2 379.2742} C_DIS
LIN {X 42.0005,Y 112.7798,Z 134,A 64.8793,B 24.9415,C -1.7674,E1 25.0573,E2 381.2358} C_DIS
LIN {X 46.1053,Y 111.165,Z 134,A 62.8629,B 24.9413,C -1.7691,E1 25.0625,E2 383.2436} C_DIS
LIN {X 49.5324,Y 109.6813,Z 134,A 61.0145,B 24.9417,C -1.7638,E1 25.0673,E2 385.0999} C_DIS
LIN {X 52.8353,Y 108.1291,Z 134,A 59.4255,B 24.9414,C -1.7686,E1 25.0712,E2 386.6735} C_DIS
LIN {X 55.4687,Y 106.8025,Z 134,A 58.0626,B 24.9414,C -1.7686,E1 25.0746,E2 388.0326} C_DIS
LIN {X 58.0301,Y 105.4339,Z 134,A 56.6082,B 24.9417,C -1.7634,E1 25.0782,E2 389.4952} C_DIS
LIN {X 60.6596,Y 103.9434,Z 134,A 55.0746,B 24.9422,C -1.7568,E1 25.0819,E2 391.0397} C_DIS
LIN {X 63.9358,Y 101.961,Z 134,A 53.2465,B 24.9424,C -1.7538,E1 25.0863,E2 392.8693} C_DIS
LIN {X 66.8706,Y 100.0601,Z 134,A 51.7304,B 24.9421,C -1.7581,E1 25.0898,E2 394.3702} C_DIS
LIN {X 69.3023,Y 98.3916,Z 134,A 50.1701,B 24.9427,C -1.7483,E1 25.0934,E2 395.9483} C_DIS
LIN {X 72.8916,Y 95.7632,Z 134,A 48.0637,B 24.9429,C -1.745,E1 25.0981,E2 398.0549} C_DIS
LIN {X 76.3522,Y 93.0274,Z 134,A 45.964,B 24.9432,C -1.7411,E1 25.1027,E2 400.156} C_DIS
LIN {X 79.7184,Y 90.1591,Z 134,A 43.8718,B 24.9434,C -1.7375,E1 25.1071,E2 402.2484} C_DIS
LIN {X 82.9769,Y 87.1699,Z 134,A 42.1228,B 24.9426,C -1.7501,E1 25.1106,E2 403.9604} C_DIS
LIN {X 85.104,Y 85.095,Z 134,A 40.3596,B 24.9439,C -1.7304,E1 25.1142,E2 405.7628} C_DIS
LIN {X 88.1787,Y 81.9039,Z 134,A 38.2654,B 24.9441,C -1.7264,E1 25.1182,E2 407.8574} C_DIS
LIN {X 91.1279,Y 78.6092,Z 134,A 36.1752,B 24.9444,C -1.7222,E1 25.1221,E2 409.948} C_DIS
LIN {X 93.975,Y 75.1831,Z 134,A 34.0733,B 24.9447,C -1.718,E1 25.1258,E2 412.05} C_DIS
LIN {X 96.6928,Y 71.6538,Z 134,A 32.0932,B 24.9446,C -1.7195,E1 25.1291,E2 414.0172} C_DIS
LIN {X 98.4668,Y 69.1956,Z 134,A 30.6804,B 24.9447,C -1.7173,E1 25.1314,E2 415.4284} C_DIS
LIN {X 100.1088,Y 66.7976,Z 134,A 29.2234,B 24.9452,C -1.7102,E1 25.1337,E2 416.895} C_DIS
LIN {X 102.1071,Y 63.7014,Z 134,A 27.4202,B 24.9456,C -1.7031,E1 25.1364,E2 418.7057} C_DIS
LIN {X 104.0048,Y 60.5541,Z 134,A 25.7045,B 24.9458,C -1.7,E1 25.1388,E2 420.4199} C_DIS
LIN {X 105.4575,Y 57.9875,Z 134,A 24.273,B 24.9462,C -1.6948,E1 25.1408,E2 421.8563} C_DIS
LIN {X 106.9849,Y 55.1164,Z 134,A 22.9503,B 24.9457,C -1.7015,E1 25.1424,E2 423.1563} C_DIS
LIN {X 108.2285,Y 52.6336,Z 134,A 21.5645,B 24.9462,C -1.6946,E1 25.1442,E2 424.551} C_DIS
LIN {X 109.4515,Y 50.039,Z 134,A 20.0982,B 24.9467,C -1.6857,E1 25.1459,E2 426.0302} C_DIS
LIN {X 111.1582,Y 46.1216,Z 134,A 18.1739,B 24.9467,C -1.6851,E1 25.148,E2 427.9453} C_DIS
LIN {X 112.2844,Y 43.308,Z 134,A 16.7566,B 24.947,C -1.6821,E1 25.1495,E2 429.3619} C_DIS
LIN {X 113.3277,Y 40.4998,Z 134,A 15.2023,B 24.9476,C -1.6716,E1 25.151,E2 430.9323} C_DIS
LIN {X 114.6181,Y 36.6878,Z 134,A 13.3617,B 24.9478,C -1.6694,E1 25.1526,E2 432.7676} C_DIS
LIN {X 115.5894,Y 33.5036,Z 134,A 11.8652,B 24.9478,C -1.6688,E1 25.1537,E2 434.2569} C_DIS
LIN {X 116.4233,Y 30.483,Z 134,A 10.283,B 24.9484,C -1.6598,E1 25.1549,E2 435.8514} C_DIS
LIN {X 117.1082,Y 27.7348,Z 134,A 9.0471,B 24.9483,C -1.6611,E1 25.1557,E2 437.0771} C_DIS
LIN {X 117.7471,Y 24.884,Z 134,A 7.667,B 24.9485,C -1.6572,E1 25.1565,E2 438.4583} C_DIS
LIN {X 118.3188,Y 22.008,Z 134,A 6.2831,B 24.9488,C -1.6533,E1 25.1573,E2 439.8432} C_DIS
LIN {X 118.8278,Y 19.0718,Z 134,A 4.8718,B 24.949,C -1.6492,E1 25.1579,E2 441.2561} C_DIS
LIN {X 119.2587,Y 16.155,Z 134,A 3.2808,B 24.9499,C -1.6354,E1 25.1585,E2 442.87} C_DIS
LIN {X 119.7841,Y 11.6249,Z 134,A 1.323,B 24.9497,C -1.6389,E1 25.1591,E2 444.8081} C_DIS
LIN {X 120.0269,Y 8.7706,Z 134,A -0.1701,B 24.9503,C -1.6281,E1 25.1595,E2 446.3177} C_DIS
LIN {X 120.2638,Y 4.4767,Z 134,A -2.0753,B 24.9503,C -1.6284,E1 25.1597,E2 448.2109} C_DIS
LIN {X 120.3404,Y 1.3968,Z 134,A -3.4685,B 24.9503,C -1.6272,E1 25.1597,E2 449.5986} C_DIS
LIN {X 120.339,Y -1.4781,Z 134,A -4.9226,B 24.9509,C -1.6185,E1 25.1597,E2 451.0646} C_DIS
LIN {X 120.264,Y -4.4723,Z 134,A -6.4801,B 24.9516,C -1.6074,E1 25.1597,E2 452.639} C_DIS
LIN {X 120.0161,Y -8.9175,Z 134,A -8.517,B 24.9518,C -1.6045,E1 25.1593,E2 454.6707} C_DIS
LIN {X 119.611,Y -13.2941,Z 134,A -10.4815,B 24.9518,C -1.6039,E1 25.1587,E2 456.6249} C_DIS
LIN {X 119.2456,Y -16.2551,Z 134,A -12.0386,B 24.9525,C -1.5925,E1 25.1581,E2 458.1997} C_DIS
LIN {X 118.8138,Y -19.1588,Z 134,A -13.3083,B 24.9524,C -1.5942,E1 25.1576,E2 459.4579} C_DIS
LIN {X 118.3043,Y -22.084,Z 134,A -14.6984,B 24.9526,C -1.5908,E1 25.1569,E2 460.848} C_DIS
LIN {X 117.7286,Y -24.9699,Z 134,A -16.093,B 24.9528,C -1.5866,E1 25.1561,E2 462.2444} C_DIS
LIN {X 117.0889,Y -27.8148,Z 134,A -17.4795,B 24.9531,C -1.5821,E1 25.1553,E2 463.6334} C_DIS
LIN {X 116.3607,Y -30.7177,Z 134,A -19.0268,B 24.9537,C -1.5715,E1 25.1542,E2 465.1967} C_DIS
LIN {X 115.167,Y -34.9277,Z 134,A -20.9656,B 24.9537,C -1.5719,E1 25.1527,E2 467.1235} C_DIS
LIN {X 114.2563,Y -37.7999,Z 134,A -22.3583,B 24.9539,C -1.5694,E1 25.1515,E2 468.5141} C_DIS
LIN {X 113.2957,Y -40.5886,Z 134,A -23.8574,B 24.9544,C -1.5603,E1 25.1501,E2 470.0264} C_DIS
LIN {X 112.2756,Y -43.3306,Z 134,A -25.1504,B 24.9544,C -1.5608,E1 25.1488,E2 471.3109} C_DIS
LIN {X 111.1615,Y -46.1136,Z 134,A -26.686,B 24.9549,C -1.551,E1 25.1471,E2 472.8611} C_DIS
LIN {X 110.0189,Y -48.7778,Z 134,A -27.9342,B 24.9548,C -1.5533,E1 25.1458,E2 474.0972} C_DIS
LIN {X 108.5519,Y -51.9592,Z 134,A -29.4401,B 24.9546,C -1.5561,E1 25.144,E2 475.5882} C_DIS
LIN {X 107.4807,Y -54.1425,Z 134,A -30.7378,B 24.9552,C -1.5457,E1 25.1424,E2 476.9037} C_DIS
LIN {X 106.0113,Y -56.9676,Z 134,A -32.1811,B 24.9552,C -1.5447,E1 25.1405,E2 478.3417} C_DIS
LIN {X 104.712,Y -59.3232,Z 134,A -33.5334,B 24.9557,C -1.5374,E1 25.1386,E2 479.7042} C_DIS
LIN {X 102.8217,Y -62.5419,Z 134,A -35.4475,B 24.9564,C -1.5254,E1 25.1359,E2 481.6367} C_DIS
LIN {X 100.8755,Y -65.6343,Z 134,A -37.022,B 24.9562,C -1.5285,E1 25.1335,E2 483.196} C_DIS
LIN {X 99.2355,Y -68.0883,Z 134,A -38.4157,B 24.9564,C -1.5251,E1 25.1313,E2 484.5909} C_DIS
LIN {X 97.101,Y -71.0995,Z 134,A -40.3262,B 24.9571,C -1.5127,E1 25.1282,E2 486.5214} C_DIS
LIN {X 94.3991,Y -74.6501,Z 134,A -42.4348,B 24.9574,C -1.5076,E1 25.1246,E2 488.6319} C_DIS
LIN {X 91.5942,Y -78.0655,Z 134,A -44.53,B 24.9577,C -1.5025,E1 25.1208,E2 490.7296} C_DIS
LIN {X 88.6428,Y -81.4012,Z 134,A -46.6241,B 24.9579,C -1.4983,E1 25.1169,E2 492.8244} C_DIS
LIN {X 85.613,Y -84.5827,Z 134,A -48.7154,B 24.9582,C -1.493,E1 25.1128,E2 494.9191} C_DIS
LIN {X 82.4513,Y -87.667,Z 134,A -50.8153,B 24.9585,C -1.488,E1 25.1086,E2 497.0221} C_DIS
LIN {X 79.1537,Y -90.6553,Z 134,A -52.9172,B 24.9588,C -1.4839,E1 25.1042,E2 499.1254} C_DIS
LIN {X 75.7726,Y -93.5002,Z 134,A -55.0018,B 24.959,C -1.48,E1 25.0997,E2 501.2111} C_DIS
LIN {X 72.3097,Y -96.2032,Z 134,A -56.7878,B 24.9584,C -1.4902,E1 25.0958,E2 502.9665} C_DIS
LIN {X 70.453,Y -97.5711,Z 134,A -58.0293,B 24.9589,C -1.481,E1 25.093,E2 504.2254} C_DIS
LIN {X 68.042,Y -99.2673,Z 134,A -59.5074,B 24.9593,C -1.4745,E1 25.0896,E2 505.7139} C_DIS
LIN {X 65.5897,Y -100.9044,Z 134,A -60.8069,B 24.9591,C -1.4767,E1 25.0866,E2 507.0038} C_DIS
LIN {X 63.0981,Y -102.4811,Z 134,A -62.2009,B 24.9593,C -1.4744,E1 25.0833,E2 508.3986} C_DIS
LIN {X 60.3939,Y -104.0975,Z 134,A -63.6553,B 24.9593,C -1.4738,E1 25.0798,E2 509.85} C_DIS
LIN {X 57.9859,Y -105.4584,Z 134,A -65.1909,B 24.96,C -1.461,E1 25.076,E2 511.4115} C_DIS
LIN {X 55.3496,Y -106.865,Z 134,A -66.4498,B 24.9597,C -1.4663,E1 25.0729,E2 512.6542} C_DIS
LIN {X 52.704,Y -108.1938,Z 134,A -67.8522,B 24.9598,C -1.4643,E1 25.0694,E2 514.0575} C_DIS
LIN {X 49.8221,Y -109.5518,Z 134,A -69.3633,B 24.9599,C -1.4622,E1 25.0656,E2 515.57} C_DIS
LIN {X 46.8988,Y -110.8336,Z 134,A -70.7985,B 24.9599,C -1.4639,E1 25.0619,E2 516.9975} C_DIS
LIN {X 44.5708,Y -111.7896,Z 134,A -72.0589,B 24.9601,C -1.4592,E1 25.0586,E2 518.2662} C_DIS
LIN {X 41.9233,Y -112.8087,Z 134,A -73.4202,B 24.9602,C -1.4569,E1 25.0551,E2 519.6301} C_DIS
LIN {X 39.1458,Y -113.8024,Z 134,A -74.8143,B 24.9603,C -1.4555,E1 25.0514,E2 521.0246} C_DIS
LIN {X 35.7635,Y -114.9112,Z 134,A -76.4326,B 24.9603,C -1.457,E1 25.0471,E2 522.6363} C_DIS
LIN {X 33.4957,Y -115.5917,Z 134,A -77.627,B 24.9605,C -1.4526,E1 25.0439,E2 523.8392} C_DIS
LIN {X 30.6585,Y -116.3765,Z 134,A -79.0288,B 24.9605,C -1.451,E1 25.0401,E2 525.2424} C_DIS
LIN {X 27.0635,Y -117.2645,Z 134,A -80.9279,B 24.961,C -1.4429,E1 25.0349,E2 527.158} C_DIS
LIN {X 23.4571,Y -118.0398,Z 134,A -82.5306,B 24.9607,C -1.4485,E1 25.0306,E2 528.7455} C_DIS
LIN {X 20.0429,Y -118.6662,Z 134,A -84.0359,B 24.9604,C -1.4541,E1 25.0265,E2 530.2358} C_DIS
LIN {X 17.6139,Y -119.0523,Z 134,A -85.365,B 24.9608,C -1.4458,E1 25.0227,E2 531.5833} C_DIS
LIN {X 14.672,Y -119.4498,Z 134,A -86.8958,B 24.9612,C -1.4394,E1 25.0185,E2 533.128} C_DIS
LIN {X 11.7587,Y -119.7713,Z 134,A -88.1668,B 24.9609,C -1.4444,E1 25.015,E2 534.3863} C_DIS
LIN {X 8.8387,Y -120.0219,Z 134,A -89.6782,B 24.9612,C -1.4384,E1 25.0107,E2 535.9114} C_DIS
LIN {X 4.4264,Y -120.2658,Z 134,A -91.652,B 24.961,C -1.4436,E1 25.0053,E2 537.8721} C_DIS
LIN {X 0.8409,Y -120.3437,Z 134,A -92.6351,B 24.9591,C -1.4769,E1 25.0027,E2 538.7761} C_DIS
Enddeposition()
LIN {X 0.8935,Y -125.788,Z 135,A -92.7847,B 24.9642,C -1.3822,E1 25.0017,E2 539.15} C_DIS
Startdeposition()
$VEL.CP = VEL_PRINT
LIN {X -1.135,Y -125.7893,Z 135,A -94.2367,B 24.9656,C -1.3561,E1 24.9975,E2 540.6639} C_DIS
LIN {X -5.0063,Y -125.694,Z 135,A -95.8483,B 24.9652,C -1.3633,E1 24.993,E2 542.2587} C_DIS
LIN {X -7.9205,Y -125.5441,Z 135,A -97.1318,B 24.9651,C -1.3655,E1 24.9894,E2 543.5374} C_DIS
LIN {X -10.789,Y -125.3302,Z 135,A -98.5248,B 24.9653,C -1.3615,E1 24.9855,E2 544.9405} C_DIS
LIN {X -14.8222,Y -124.9172,Z 135,A -100.3676,B 24.9653,C -1.3619,E1 24.9804,E2 546.7834} C_DIS
LIN {X -17.9993,Y -124.4992,Z 135,A -101.7901,B 24.9652,C -1.364,E1 24.9765,E2 548.2021} C_DIS
LIN {X -20.7354,Y -124.0727,Z 135,A -103.0839,B 24.9652,C -1.3628,E1 24.9729,E2 549.4998} C_DIS
LIN {X -24.0617,Y -123.4715,Z 135,A -104.5674,B 24.965,C -1.3661,E1 24.9689,E2 550.9772} C_DIS
LIN {X -27.0207,Y -122.858,Z 135,A -105.9535,B 24.965,C -1.3662,E1 24.9651,E2 552.3646} C_DIS
LIN {X -29.6758,Y -122.243,Z 135,A -107.2831,B 24.9652,C -1.3627,E1 24.9614,E2 553.7044} C_DIS
LIN {X -32.8456,Y -121.4303,Z 135,A -108.682,B 24.9649,C -1.368,E1 24.9577,E2 555.0928} C_DIS
LIN {X -35.4912,Y -120.6828,Z 135,A -109.9812,B 24.965,C -1.3666,E1 24.9542,E2 556.3974} C_DIS
LIN {X -38.4734,Y -119.7655,Z 135,A -111.4002,B 24.965,C -1.3678,E1 24.9504,E2 557.8161} C_DIS
LIN {X -41.4108,Y -118.7818,Z 135,A -112.8203,B 24.965,C -1.3685,E1 24.9466,E2 559.2371} C_DIS
LIN {X -44.8513,Y -117.5282,Z 135,A -114.4863,B 24.9648,C -1.3701,E1 24.9423,E2 560.9028} C_DIS
LIN {X -47.3132,Y -116.5567,Z 135,A -115.7419,B 24.9648,C -1.369,E1 24.939,E2 562.1638} C_DIS
LIN {X -50.1247,Y -115.3754,Z 135,A -117.1056,B 24.9648,C -1.3717,E1 24.9355,E2 563.5243} C_DIS
LIN {X -53.5129,Y -113.8459,Z 135,A -118.7888,B 24.9646,C -1.3741,E1 24.9313,E2 565.2059} C_DIS
LIN {X -56.3617,Y -112.4628,Z 135,A -120.2569,B 24.9646,C -1.3747,E1 24.9276,E2 566.6765} C_DIS
LIN {X -59.8882,Y -110.6251,Z 135,A -122.2133,B 24.9648,C -1.3703,E1 24.9227,E2 568.6488} C_DIS
LIN {X -63.9272,Y -108.3409,Z 135,A -124.2718,B 24.9645,C -1.3759,E1 24.9177,E2 570.7001} C_DIS
LIN {X -67.4834,Y -106.1627,Z 135,A -126.1107,B 24.9642,C -1.3816,E1 24.9134,E2 572.531} C_DIS
LIN {X -70.8068,Y -103.9754,Z 135,A -128.0076,B 24.9642,C -1.3807,E1 24.909,E2 574.4366} C_DIS
LIN {X -74.1429,Y -101.6236,Z 135,A -129.8914,B 24.9642,C -1.3827,E1 24.9047,E2 576.3221} C_DIS
LIN {X -77.5034,Y -99.084,Z 135,A -131.8225,B 24.964,C -1.3856,E1 24.9004,E2 578.2532} C_DIS
LIN {X -80.9421,Y -96.2952,Z 135,A -133.8187,B 24.9638,C -1.3904,E1 24.8961,E2 580.2457} C_DIS
LIN {X -84.2174,Y -93.4448,Z 135,A -135.8507,B 24.9638,C -1.3919,E1 24.8919,E2 582.2822} C_DIS
LIN {X -87.4174,Y -90.4576,Z 135,A -137.8035,B 24.9634,C -1.398,E1 24.8879,E2 584.2286} C_DIS
LIN {X -90.5358,Y -87.3366,Z 135,A -139.8308,B 24.9632,C -1.4015,E1 24.884,E2 586.2561} C_DIS
LIN {X -93.4343,Y -84.2293,Z 135,A -141.8003,B 24.9631,C -1.4043,E1 24.8802,E2 588.2276} C_DIS
LIN {X -96.2318,Y -81.0176,Z 135,A -143.7401,B 24.9628,C -1.4089,E1 24.8767,E2 590.1654} C_DIS
LIN {X -98.9979,Y -77.6131,Z 135,A -145.6752,B 24.9624,C -1.4166,E1 24.8734,E2 592.0912} C_DIS
LIN {X -101.2794,Y -74.6115,Z 135,A -147.4621,B 24.9624,C -1.4177,E1 24.8704,E2 593.884} C_DIS
LIN {X -103.7831,Y -71.0875,Z 135,A -149.4233,B 24.9621,C -1.4231,E1 24.8672,E2 595.842} C_DIS
LIN {X -106.1627,Y -67.4834,Z 135,A -151.3954,B 24.9618,C -1.4281,E1 24.8642,E2 597.8123} C_DIS
LIN {X -108.3008,Y -63.9954,Z 135,A -153.3299,B 24.9618,C -1.4299,E1 24.8614,E2 599.7524} C_DIS
LIN {X -110.5882,Y -59.956,Z 135,A -155.4278,B 24.9613,C -1.4365,E1 24.8586,E2 601.8457} C_DIS
LIN {X -112.2571,Y -56.7657,Z 135,A -157.0008,B 24.9609,C -1.4441,E1 24.8566,E2 603.4089} C_DIS
LIN {X -113.7816,Y -53.6475,Z 135,A -158.5351,B 24.9606,C -1.4507,E1 24.8548,E2 604.9357} C_DIS
LIN {X -115.1513,Y -50.6428,Z 135,A -160.0607,B 24.9604,C -1.4541,E1 24.853,E2 606.4616} C_DIS
LIN {X -116.1401,Y -48.3261,Z 135,A -161.2223,B 24.9602,C -1.4569,E1 24.8518,E2 607.6231} C_DIS
LIN {X -117.3463,Y -45.3192,Z 135,A -162.689,B 24.96,C -1.4617,E1 24.8503,E2 609.0866} C_DIS
LIN {X -118.4107,Y -42.4602,Z 135,A -164.0999,B 24.9598,C -1.4649,E1 24.8489,E2 610.4978} C_DIS
LIN {X -119.5937,Y -39.0113,Z 135,A -165.7635,B 24.9595,C -1.4697,E1 24.8474,E2 612.1593} C_DIS
LIN {X -120.7854,Y -35.1408,Z 135,A -167.6729,B 24.9594,C -1.4725,E1 24.8459,E2 614.0731} C_DIS
LIN {X -121.9471,Y -30.8685,Z 135,A -169.667,B 24.959,C -1.4798,E1 24.8445,E2 616.0613} C_DIS
LIN {X -122.6411,Y -27.9843,Z 135,A -171.0349,B 24.9588,C -1.4833,E1 24.8436,E2 617.4289} C_DIS
LIN {X -123.2851,Y -24.9954,Z 135,A -172.4225,B 24.9585,C -1.488,E1 24.8428,E2 618.8138} C_DIS
LIN {X -123.8991,Y -21.7521,Z 135,A -173.9381,B 24.9583,C -1.4922,E1 24.842,E2 620.3282} C_DIS
LIN {X -124.4182,Y -18.5625,Z 135,A -175.3899,B 24.958,C -1.4978,E1 24.8414,E2 621.7753} C_DIS
LIN {X -124.8217,Y -15.6225,Z 135,A -176.9099,B 24.9581,C -1.4946,E1 24.8409,E2 623.3119} C_DIS
LIN {X -125.2228,Y -11.9695,Z 135,A -178.4355,B 24.9575,C -1.5067,E1 24.8404,E2 624.8179} C_DIS
LIN {X -125.4743,Y -8.9583,Z 135,A -179.8713,B 24.9574,C -1.5085,E1 24.8401,E2 626.258} C_DIS
LIN {X -125.6588,Y -5.84,Z 135,A 178.7701,B 24.9569,C -1.516,E1 24.8399,E2 627.6069} C_DIS
LIN {X -125.7716,Y -2.3721,Z 135,A 177.0836,B 24.9569,C -1.5165,E1 24.8398,E2 629.3025} C_DIS
LIN {X -125.7795,Y 1.8958,Z 135,A 175.1321,B 24.9566,C -1.5225,E1 24.8398,E2 631.2514} C_DIS
LIN {X -125.6705,Y 5.608,Z 135,A 173.4985,B 24.9561,C -1.5306,E1 24.84,E2 632.8755} C_DIS
LIN {X -125.4604,Y 9.1493,Z 135,A 171.8289,B 24.9559,C -1.5335,E1 24.8403,E2 634.5482} C_DIS
LIN {X -125.1726,Y 12.4924,Z 135,A 170.349,B 24.9555,C -1.5407,E1 24.8407,E2 636.0198} C_DIS
LIN {X -124.8836,Y 15.1037,Z 135,A 169.0651,B 24.9555,C -1.5407,E1 24.8411,E2 637.3113} C_DIS
LIN {X -124.2933,Y 19.3697,Z 135,A 167.1516,B 24.955,C -1.5493,E1 24.8418,E2 639.2158} C_DIS
LIN {X -123.7893,Y 22.3658,Z 135,A 165.7576,B 24.9548,C -1.5534,E1 24.8425,E2 640.6085} C_DIS
LIN {X -123.1811,Y 25.5063,Z 135,A 164.2516,B 24.9546,C -1.5559,E1 24.8433,E2 642.1172} C_DIS
LIN {X -122.5877,Y 28.2182,Z 135,A 162.9481,B 24.9546,C -1.5583,E1 24.8441,E2 643.4227} C_DIS
LIN {X -121.8959,Y 31.0703,Z 135,A 161.6245,B 24.9542,C -1.5632,E1 24.845,E2 644.7424} C_DIS
LIN {X -121.1396,Y 33.8989,Z 135,A 160.2812,B 24.954,C -1.5671,E1 24.846,E2 646.0843} C_DIS
LIN {X -120.2228,Y 37.0197,Z 135,A 158.7908,B 24.9537,C -1.5714,E1 24.8472,E2 647.5729} C_DIS
LIN {X -119.3054,Y 39.8769,Z 135,A 157.422,B 24.9535,C -1.5757,E1 24.8484,E2 648.9395} C_DIS
LIN {X -118.2237,Y 42.9788,Z 135,A 155.8855,B 24.9533,C -1.5786,E1 24.8498,E2 650.4777} C_DIS
LIN {X -116.5773,Y 47.2621,Z 135,A 153.7637,B 24.953,C -1.5837,E1 24.852,E2 652.5992} C_DIS
LIN {X -114.7394,Y 51.5638,Z 135,A 151.6596,B 24.9525,C -1.5915,E1 24.8543,E2 654.6964} C_DIS
LIN {X -113.1834,Y 54.8996,Z 135,A 149.9828,B 24.9522,C -1.5965,E1 24.8563,E2 656.3702} C_DIS
LIN {X -111.9576,Y 57.354,Z 135,A 148.6792,B 24.9522,C -1.5979,E1 24.858,E2 657.6775} C_DIS
LIN {X -110.4879,Y 60.1399,Z 135,A 147.1884,B 24.9521,C -1.5997,E1 24.86,E2 659.172} C_DIS
LIN {X -108.3707,Y 63.8764,Z 135,A 145.2036,B 24.9518,C -1.6041,E1 24.8627,E2 661.1566} C_DIS
LIN {X -106.1627,Y 67.4834,Z 135,A 143.2492,B 24.9515,C -1.6084,E1 24.8656,E2 663.1107} C_DIS
LIN {X -103.9473,Y 70.8483,Z 135,A 141.4271,B 24.9512,C -1.6142,E1 24.8684,E2 664.9281} C_DIS
LIN {X -101.6182,Y 74.1503,Z 135,A 139.5489,B 24.951,C -1.6176,E1 24.8715,E2 666.8073} C_DIS
LIN {X -99.178,Y 77.3838,Z 135,A 137.7032,B 24.9507,C -1.6226,E1 24.8746,E2 668.6498} C_DIS
LIN {X -96.6461,Y 80.5235,Z 135,A 135.8405,B 24.9504,C -1.6264,E1 24.8779,E2 670.5123} C_DIS
LIN {X -93.977,Y 83.6232,Z 135,A 133.9805,B 24.9501,C -1.6313,E1 24.8814,E2 672.3688} C_DIS
LIN {X -91.2235,Y 86.6187,Z 135,A 132.1515,B 24.9498,C -1.6371,E1 24.8848,E2 674.192} C_DIS
LIN {X -88.3733,Y 89.5247,Z 135,A 130.3098,B 24.9495,C -1.6422,E1 24.8885,E2 676.0294} C_DIS
LIN {X -85.431,Y 92.3367,Z 135,A 128.4247,B 24.9493,C -1.6453,E1 24.8923,E2 677.9151} C_DIS
LIN {X -82.4011,Y 95.0504,Z 135,A 126.5988,B 24.9489,C -1.6508,E1 24.8961,E2 679.735} C_DIS
LIN {X -79.2887,Y 97.6618,Z 135,A 124.6592,B 24.9489,C -1.6508,E1 24.9003,E2 681.6818} C_DIS
LIN {X -76.099,Y 100.1672,Z 135,A 122.7779,B 24.9488,C -1.6533,E1 24.9044,E2 683.5642} C_DIS
LIN {X -72.6001,Y 102.7307,Z 135,A 120.8499,B 24.9484,C -1.6596,E1 24.9088,E2 685.4839} C_DIS
LIN {X -69.2677,Y 105.0065,Z 135,A 119.0053,B 24.9482,C -1.6629,E1 24.9131,E2 687.3267} C_DIS
LIN {X -65.6827,Y 107.2854,Z 135,A 117.0591,B 24.948,C -1.6661,E1 24.9177,E2 689.2715} C_DIS
LIN {X -61.9964,Y 109.4576,Z 135,A 115.0506,B 24.948,C -1.6669,E1 24.9225,E2 691.2841} C_DIS
LIN {X -58.2836,Y 111.4763,Z 135,A 113.2585,B 24.9473,C -1.6763,E1 24.9269,E2 693.0588} C_DIS
LIN {X -54.9402,Y 113.1641,Z 135,A 111.5595,B 24.9471,C -1.6794,E1 24.9312,E2 694.755} C_DIS
LIN {X -52.4952,Y 114.3165,Z 135,A 110.2923,B 24.9471,C -1.6797,E1 24.9344,E2 696.0246} C_DIS
LIN {X -49.5534,Y 115.6224,Z 135,A 108.8771,B 24.9468,C -1.6842,E1 24.938,E2 697.4325} C_DIS
LIN {X -46.8257,Y 116.7532,Z 135,A 107.5264,B 24.9468,C -1.6859,E1 24.9415,E2 698.7822} C_DIS
LIN {X -43.9183,Y 117.8777,Z 135,A 106.0869,B 24.9467,C -1.6869,E1 24.9452,E2 700.2224} C_DIS
LIN {X -40.7956,Y 118.9951,Z 135,A 104.5488,B 24.9467,C -1.6875,E1 24.9493,E2 701.7619} C_DIS
LIN {X -36.548,Y 120.3672,Z 135,A 102.5469,B 24.9464,C -1.6914,E1 24.9546,E2 703.7583} C_DIS
LIN {X -33.1464,Y 121.3501,Z 135,A 100.9239,B 24.9464,C -1.6926,E1 24.959,E2 705.3809} C_DIS
LIN {X -29.272,Y 122.3403,Z 135,A 99.0881,B 24.9462,C -1.6937,E1 24.9639,E2 707.2167} C_DIS
LIN {X -26.476,Y 122.9756,Z 135,A 97.7719,B 24.9462,C -1.6944,E1 24.9675,E2 708.5328} C_DIS
LIN {X -23.4152,Y 123.5951,Z 135,A 96.3517,B 24.9462,C -1.6957,E1 24.9714,E2 709.9516} C_DIS
LIN {X -19.9745,Y 124.1996,Z 135,A 94.7812,B 24.946,C -1.6978,E1 24.9757,E2 711.5186} C_DIS
LIN {X -17.5159,Y 124.5683,Z 135,A 93.6064,B 24.946,C -1.6966,E1 24.979,E2 712.6972} C_DIS
LIN {X -13.8183,Y 125.0327,Z 135,A 91.8707,B 24.9461,C -1.6958,E1 24.9838,E2 714.4361} C_DIS
LIN {X -10.5739,Y 125.3483,Z 135,A 90.4364,B 24.9459,C -1.6989,E1 24.9878,E2 715.8637} C_DIS
LIN {X -7.2066,Y 125.5881,Z 135,A 88.9474,B 24.9457,C -1.7018,E1 24.9919,E2 717.3463} C_DIS
LIN {X -4.7042,Y 125.7058,Z 135,A 87.7392,B 24.9459,C -1.699,E1 24.9953,E2 718.5613} C_DIS
LIN {X -0.8924,Y 125.7906,Z 135,A 85.9787,B 24.9459,C -1.6983,E1 25.0002,E2 720.3236} C_DIS
LIN {X 2.1801,Y 125.7748,Z 135,A 84.58,B 24.9459,C -1.6986,E1 25.0041,E2 721.7216} C_DIS
LIN {X 6.1789,Y 125.6418,Z 135,A 82.7635,B 24.9459,C -1.699,E1 25.0092,E2 723.5366} C_DIS
LIN {X 9.1182,Y 125.4626,Z 135,A 81.4414,B 24.9459,C -1.6998,E1 25.0129,E2 724.8561} C_DIS
LIN {X 12.5996,Y 125.1623,Z 135,A 79.9145,B 24.9457,C -1.7028,E1 25.0171,E2 726.3752} C_DIS
LIN {X 15.0711,Y 124.8875,Z 135,A 78.6949,B 24.9459,C -1.6984,E1 25.0205,E2 727.6042} C_DIS
LIN {X 19.3976,Y 124.2889,Z 135,A 76.7963,B 24.9457,C -1.7022,E1 25.0257,E2 729.4921} C_DIS
LIN {X 22.3482,Y 123.7924,Z 135,A 75.4213,B 24.9457,C -1.7011,E1 25.0295,E2 730.8682} C_DIS
LIN {X 25.2563,Y 123.232,Z 135,A 73.9878,B 24.9461,C -1.6964,E1 25.0334,E2 732.311} C_DIS
LIN {X 29.702,Y 122.2366,Z 135,A 71.9209,B 24.9461,C -1.6957,E1 25.0391,E2 734.3768} C_DIS
LIN {X 34.0584,Y 121.095,Z 135,A 69.8728,B 24.9461,C -1.6945,E1 25.0446,E2 736.4245} C_DIS
LIN {X 37.0197,Y 120.2228,Z 135,A 68.5386,B 24.9461,C -1.6969,E1 25.0481,E2 737.7506} C_DIS
LIN {X 39.9487,Y 119.2815,Z 135,A 67.1183,B 24.9461,C -1.6948,E1 25.0519,E2 739.1731} C_DIS
LIN {X 42.8855,Y 118.2574,Z 135,A 65.6455,B 24.9464,C -1.6908,E1 25.0558,E2 740.6525} C_DIS
LIN {X 45.7824,Y 117.1663,Z 135,A 64.286,B 24.9464,C -1.6919,E1 25.0593,E2 742.0066} C_DIS
LIN {X 49.2008,Y 115.7748,Z 135,A 62.6155,B 24.9464,C -1.6905,E1 25.0636,E2 743.6763} C_DIS
LIN {X 51.6096,Y 114.7189,Z 135,A 61.3668,B 24.9467,C -1.6867,E1 25.0668,E2 744.931} C_DIS
LIN {X 54.573,Y 113.3394,Z 135,A 59.8984,B 24.9467,C -1.6859,E1 25.0705,E2 746.3975} C_DIS
LIN {X 57.5983,Y 111.8333,Z 135,A 58.3869,B 24.9467,C -1.6852,E1 25.0743,E2 747.9065} C_DIS
LIN {X 60.8534,Y 110.0965,Z 135,A 56.6327,B 24.9472,C -1.6792,E1 25.0786,E2 749.6698} C_DIS
LIN {X 64.309,Y 108.1144,Z 135,A 54.8034,B 24.9474,C -1.6758,E1 25.083,E2 751.5016} C_DIS
LIN {X 68.1551,Y 105.7327,Z 135,A 52.7718,B 24.9474,C -1.674,E1 25.0878,E2 753.531} C_DIS
LIN {X 71.5805,Y 103.4442,Z 135,A 50.848,B 24.9478,C -1.6685,E1 25.0923,E2 755.4613} C_DIS
LIN {X 75.2188,Y 100.8291,Z 135,A 48.9059,B 24.9478,C -1.6698,E1 25.0966,E2 757.3935} C_DIS
LIN {X 78.1484,Y 98.5761,Z 135,A 47.1488,B 24.9482,C -1.663,E1 25.1005,E2 759.1601} C_DIS
LIN {X 81.6791,Y 95.6711,Z 135,A 45.1063,B 24.9483,C -1.6609,E1 25.1049,E2 761.1997} C_DIS
LIN {X 84.8318,Y 92.8875,Z 135,A 43.1691,B 24.9486,C -1.6559,E1 25.1089,E2 763.1409} C_DIS
LIN {X 87.7921,Y 90.0948,Z 135,A 41.3685,B 24.9486,C -1.6546,E1 25.1126,E2 764.9371} C_DIS
LIN {X 90.6611,Y 87.2072,Z 135,A 39.5231,B 24.9489,C -1.651,E1 25.1162,E2 766.7833} C_DIS
LIN {X 93.4343,Y 84.2293,Z 135,A 37.6173,B 24.9493,C -1.6441,E1 25.1198,E2 768.6968} C_DIS
LIN {X 96.237,Y 81.0113,Z 135,A 35.713,B 24.9495,C -1.6415,E1 25.1232,E2 770.5986} C_DIS
LIN {X 98.9979,Y 77.6131,Z 135,A 33.7943,B 24.9495,C -1.6405,E1 25.1266,E2 772.5108} C_DIS
LIN {X 101.4963,Y 74.3162,Z 135,A 31.8667,B 24.95,C -1.6335,E1 25.1298,E2 774.4455} C_DIS
LIN {X 103.9473,Y 70.8483,Z 135,A 29.9664,B 24.9502,C -1.6303,E1 25.1328,E2 776.3442} C_DIS
LIN {X 106.1627,Y 67.4834,Z 135,A 28.1458,B 24.9505,C -1.6261,E1 25.1356,E2 778.1654} C_DIS
LIN {X 108.2911,Y 64.0118,Z 135,A 26.2276,B 24.951,C -1.6179,E1 25.1384,E2 780.0933} C_DIS
LIN {X 110.5725,Y 59.9848,Z 135,A 24.1593,B 24.9512,C -1.6141,E1 25.1412,E2 782.1598} C_DIS
LIN {X 112.2038,Y 56.8704,Z 135,A 22.6903,B 24.951,C -1.6164,E1 25.143,E2 783.6156} C_DIS
LIN {X 113.5895,Y 54.0497,Z 135,A 21.2588,B 24.9513,C -1.6122,E1 25.1448,E2 785.0491} C_DIS
LIN {X 115.1513,Y 50.6428,Z 135,A 19.5737,B 24.9515,C -1.6084,E1 25.1467,E2 786.7342} C_DIS
LIN {X 116.1268,Y 48.3581,Z 135,A 18.4364,B 24.9517,C -1.6048,E1 25.1479,E2 787.8738} C_DIS
LIN {X 117.3495,Y 45.3112,Z 135,A 16.9755,B 24.9519,C -1.6021,E1 25.1494,E2 789.3329} C_DIS
LIN {X 118.4071,Y 42.4703,Z 135,A 15.5752,B 24.9522,C -1.5969,E1 25.1508,E2 790.7375} C_DIS
LIN {X 119.5937,Y 39.0113,Z 135,A 13.9431,B 24.9524,C -1.5935,E1 25.1522,E2 792.3684} C_DIS
LIN {X 120.4058,Y 36.4218,Z 135,A 12.7381,B 24.9526,C -1.5914,E1 25.1532,E2 793.5717} C_DIS
LIN {X 121.3501,Y 33.1464,Z 135,A 11.1765,B 24.9529,C -1.586,E1 25.1544,E2 795.1368} C_DIS
LIN {X 122.3403,Y 29.272,Z 135,A 9.3549,B 24.9532,C -1.5804,E1 25.1556,E2 796.9614} C_DIS
LIN {X 122.9609,Y 26.5439,Z 135,A 8.0695,B 24.9535,C -1.5758,E1 25.1564,E2 798.2501} C_DIS
LIN {X 123.5951,Y 23.4152,Z 135,A 6.6541,B 24.9536,C -1.5731,E1 25.1572,E2 799.6634} C_DIS
LIN {X 124.1901,Y 20.0315,Z 135,A 5.1119,B 24.9539,C -1.5692,E1 25.1579,E2 801.2057} C_DIS
LIN {X 124.5898,Y 17.3656,Z 135,A 3.9223,B 24.9539,C -1.5673,E1 25.1584,E2 802.3929} C_DIS
LIN {X 124.994,Y 14.1787,Z 135,A 2.4444,B 24.9543,C -1.5618,E1 25.1589,E2 803.8751} C_DIS
LIN {X 125.3585,Y 10.454,Z 135,A 0.7444,B 24.9546,C -1.5565,E1 25.1593,E2 805.5775} C_DIS
LIN {X 125.5993,Y 7.0242,Z 135,A -0.7979,B 24.9548,C -1.5526,E1 25.1596,E2 807.1198} C_DIS
LIN {X 125.7115,Y 4.5576,Z 135,A -2.0758,B 24.9555,C -1.541,E1 25.1597,E2 808.4175} C_DIS
LIN {X 125.7953,Y 0.3519,Z 135,A -4.032,B 24.956,C -1.5326,E1 25.1597,E2 810.3818} C_DIS
LIN {X 125.7427,Y -3.5777,Z 135,A -5.6709,B 24.9559,C -1.5345,E1 25.1597,E2 812.0063} C_DIS
LIN {X 125.5432,Y -7.9349,Z 135,A -7.5363,B 24.9559,C -1.5343,E1 25.1594,E2 813.8612} C_DIS
LIN {X 125.3302,Y -10.789,Z 135,A -8.9055,B 24.9563,C -1.5266,E1 25.1591,E2 815.2404} C_DIS
LIN {X 125.0496,Y -13.6613,Z 135,A -10.1571,B 24.9563,C -1.5255,E1 25.1588,E2 816.4871} C_DIS
LIN {X 124.7358,Y -16.278,Z 135,A -11.4191,B 24.9568,C -1.5184,E1 25.1583,E2 817.7585} C_DIS
LIN {X 124.2805,Y -19.452,Z 135,A -12.7861,B 24.9568,C -1.5184,E1 25.1578,E2 819.1173} C_DIS
LIN {X 123.7893,Y -22.3658,Z 135,A -14.1742,B 24.9572,C -1.5118,E1 25.1571,E2 820.5128} C_DIS
LIN {X 123.2214,Y -25.3084,Z 135,A -15.5729,B 24.9575,C -1.5056,E1 25.1563,E2 821.9181} C_DIS
LIN {X 122.2095,Y -29.8148,Z 135,A -17.6468,B 24.9578,C -1.5003,E1 25.155,E2 823.9924} C_DIS
LIN {X 121.404,Y -32.944,Z 135,A -19.0503,B 24.9578,C -1.4991,E1 25.154,E2 825.3907} C_DIS
LIN {X 120.5103,Y -36.0805,Z 135,A -20.5524,B 24.9582,C -1.4934,E1 25.1528,E2 826.8976} C_DIS
LIN {X 119.2815,Y -39.9487,Z 135,A -22.3915,B 24.9585,C -1.4881,E1 25.1513,E2 828.739} C_DIS
LIN {X 118.2168,Y -42.9981,Z 135,A -23.8911,B 24.9589,C -1.4819,E1 25.1498,E2 830.2446} C_DIS
LIN {X 117.1663,Y -45.7824,Z 135,A -25.2319,B 24.9591,C -1.4784,E1 25.1485,E2 831.5862} C_DIS
LIN {X 115.7748,Y -49.2008,Z 135,A -26.874,B 24.9592,C -1.4752,E1 25.1467,E2 833.2269} C_DIS
LIN {X 114.7075,Y -51.635,Z 135,A -28.1253,B 24.9596,C -1.4693,E1 25.1453,E2 834.4851} C_DIS
LIN {X 113.2884,Y -54.6799,Z 135,A -29.618,B 24.9597,C -1.4666,E1 25.1435,E2 835.9764} C_DIS
LIN {X 111.7873,Y -57.6887,Z 135,A -31.201,B 24.9601,C -1.4592,E1 25.1415,E2 837.5682} C_DIS
LIN {X 109.8565,Y -61.2869,Z 135,A -33.0523,B 24.9604,C -1.4541,E1 25.139,E2 839.4219} C_DIS
LIN {X 107.8077,Y -64.8226,Z 135,A -34.9614,B 24.9608,C -1.4462,E1 25.1363,E2 841.3398} C_DIS
LIN {X 105.5712,Y -68.4039,Z 135,A -36.8269,B 24.961,C -1.4436,E1 25.1335,E2 843.2021} C_DIS
LIN {X 103.3247,Y -71.7522,Z 135,A -38.6537,B 24.9612,C -1.4389,E1 25.1306,E2 845.031} C_DIS
LIN {X 100.7509,Y -75.3238,Z 135,A -40.6424,B 24.9615,C -1.4341,E1 25.1274,E2 847.0213} C_DIS
LIN {X 98.1715,Y -78.6568,Z 135,A -42.5833,B 24.9618,C -1.4278,E1 25.124,E2 848.968} C_DIS
LIN {X 95.4949,Y -81.885,Z 135,A -44.4968,B 24.9621,C -1.4225,E1 25.1205,E2 850.8852} C_DIS
LIN {X 92.6691,Y -85.0695,Z 135,A -46.3797,B 24.9622,C -1.4204,E1 25.117,E2 852.7647} C_DIS
LIN {X 89.8899,Y -88.001,Z 135,A -48.2169,B 24.9624,C -1.4159,E1 25.1135,E2 854.6047} C_DIS
LIN {X 86.8409,Y -91.0112,Z 135,A -50.1486,B 24.9626,C -1.4121,E1 25.1096,E2 856.5372} C_DIS
LIN {X 83.6537,Y -93.9497,Z 135,A -52.1112,B 24.9629,C -1.408,E1 25.1055,E2 858.5016} C_DIS
LIN {X 80.5432,Y -96.6298,Z 135,A -53.9671,B 24.9631,C -1.4044,E1 25.1016,E2 860.3587} C_DIS
LIN {X 77.3838,Y -99.178,Z 135,A -55.8734,B 24.9634,C -1.3974,E1 25.0974,E2 862.2745} C_DIS
LIN {X 73.9149,Y -101.7888,Z 135,A -57.7899,B 24.9634,C -1.3963,E1 25.0931,E2 864.1869} C_DIS
LIN {X 70.6082,Y -104.1098,Z 135,A -59.6209,B 24.9637,C -1.393,E1 25.0889,E2 866.0194} C_DIS
LIN {X 66.9285,Y -106.5129,Z 135,A -61.6228,B 24.9639,C -1.389,E1 25.0842,E2 868.0242} C_DIS
LIN {X 63.3708,Y -108.6677,Z 135,A -63.4823,B 24.9639,C -1.3872,E1 25.0797,E2 869.8822} C_DIS
LIN {X 59.8882,Y -110.6251,Z 135,A -65.3301,B 24.9642,C -1.3825,E1 25.0752,E2 871.7357} C_DIS
LIN {X 56.7616,Y -112.2592,Z 135,A -66.859,B 24.9642,C -1.3837,E1 25.0714,E2 873.2575} C_DIS
LIN {X 53.664,Y -113.7737,Z 135,A -68.368,B 24.9642,C -1.3842,E1 25.0676,E2 874.7613} C_DIS
LIN {X 50.6428,Y -115.1513,Z 135,A -69.8885,B 24.9642,C -1.3815,E1 25.0637,E2 876.2847} C_DIS
LIN {X 48.3105,Y -116.1466,Z 135,A -71.0442,B 24.9643,C -1.3798,E1 25.0608,E2 877.4417} C_DIS
LIN {X 45.3522,Y -117.3335,Z 135,A -72.4809,B 24.9644,C -1.3784,E1 25.057,E2 878.8783} C_DIS
LIN {X 42.4602,Y -118.4107,Z 135,A -73.8909,B 24.9645,C -1.3763,E1 25.0533,E2 880.2903} C_DIS
LIN {X 39.1361,Y -119.5521,Z 135,A -75.4586,B 24.9645,C -1.3759,E1 25.0492,E2 881.8559} C_DIS
LIN {X 36.4157,Y -120.4077,Z 135,A -76.751,B 24.9646,C -1.3747,E1 25.0457,E2 883.1488} C_DIS
LIN {X 33.1464,Y -121.3501,Z 135,A -78.3166,B 24.9647,C -1.3722,E1 25.0415,E2 884.7179} C_DIS
LIN {X 29.272,Y -122.3403,Z 135,A -80.1579,B 24.9649,C -1.3694,E1 25.0365,E2 886.5631} C_DIS
LIN {X 26.4428,Y -122.9827,Z 135,A -81.4649,B 24.9649,C -1.3688,E1 25.033,E2 887.8696} C_DIS
LIN {X 23.4152,Y -123.5951,Z 135,A -82.8464,B 24.9649,C -1.3688,E1 25.0292,E2 889.2494} C_DIS
LIN {X 19.9745,Y -124.1996,Z 135,A -84.4363,B 24.9649,C -1.3677,E1 25.0248,E2 890.8404} C_DIS
LIN {X 17.4291,Y -124.5807,Z 135,A -85.5866,B 24.9649,C -1.368,E1 25.0216,E2 891.9891} C_DIS
LIN {X 14.1787,Y -124.994,Z 135,A -87.0925,B 24.965,C -1.3663,E1 25.0174,E2 893.4976} C_DIS
LIN {X 11.3033,Y -125.2867,Z 135,A -88.5717,B 24.9655,C -1.3576,E1 25.0133,E2 894.9966} C_DIS
LIN {X 7.6335,Y -125.5618,Z 135,A -90.1507,B 24.9653,C -1.3617,E1 25.0089,E2 896.5653} C_DIS
LIN {X 3.6286,Y -125.7413,Z 135,A -91.9619,B 24.9653,C -1.3617,E1 25.0038,E2 898.3759} C_DIS
LIN {X 0.8935,Y -125.788,Z 135,A -92.7846,B 24.9642,C -1.3822,E1 25.0017,E2 899.15} C_DIS
Enddeposition()
LIN {X 0.8935,Y -125.788,Z 135,A -92.7846,B 24.9642,C -1.3822,E1 25.0017,E2 899.15} C_DIS
Startdeposition()
$VEL.CP = VEL_PRINT
LIN {X 2.7365,Y -124.7726,Z 135,A -91.5737,B 24.9624,C -1.4176,E1 25.0053,E2 897.8555} C_DIS
LIN {X 6.5022,Y -124.6315,Z 135,A -89.9801,B 24.9627,C -1.4115,E1 25.0097,E2 896.2766} C_DIS
LIN {X 10.1621,Y -124.3868,Z 135,A -88.2492,B 24.9625,C -1.4147,E1 25.0145,E2 894.5392} C_DIS
LIN {X 13.9096,Y -124.0244,Z 135,A -86.6058,B 24.9627,C -1.4114,E1 25.0191,E2 892.9045} C_DIS
LIN {X 17.0617,Y -123.6303,Z 135,A -85.0594,B 24.9624,C -1.4167,E1 25.0234,E2 891.3468} C_DIS
LIN {X 20.8943,Y -123.0396,Z 135,A -83.2663,B 24.9623,C -1.4187,E1 25.0283,E2 889.5507} C_DIS
LIN {X 24.8001,Y -122.3117,Z 135,A -81.5132,B 24.9623,C -1.4168,E1 25.0331,E2 887.8043} C_DIS
LIN {X 28.0018,Y -121.6188,Z 135,A -79.9547,B 24.9622,C -1.4209,E1 25.0374,E2 886.2382} C_DIS
LIN {X 32.1749,Y -120.5817,Z 135,A -77.9877,B 24.9621,C -1.4226,E1 25.0427,E2 884.2701} C_DIS
LIN {X 37.3715,Y -119.0753,Z 135,A -75.5047,B 24.9619,C -1.4254,E1 25.0494,E2 881.7848} C_DIS
LIN {X 40.8885,Y -117.9121,Z 135,A -73.8741,B 24.962,C -1.4241,E1 25.0537,E2 880.1606} C_DIS
LIN {X 44.116,Y -116.7435,Z 135,A -72.2184,B 24.9617,C -1.4303,E1 25.058,E2 878.4938} C_DIS
LIN {X 47.6188,Y -115.3596,Z 135,A -70.6336,B 24.9619,C -1.4255,E1 25.0621,E2 876.9239} C_DIS
LIN {X 50.9388,Y -113.9314,Z 135,A -68.832,B 24.9614,C -1.4352,E1 25.0667,E2 875.1037} C_DIS
LIN {X 55.661,Y -111.7015,Z 135,A -66.3821,B 24.9611,C -1.4418,E1 25.0729,E2 872.6447} C_DIS
LIN {X 59.4475,Y -109.7347,Z 135,A -63.9597,B 24.9596,C -1.4688,E1 25.079,E2 870.1653} C_DIS
LIN {X 63.5049,Y -107.4375,Z 135,A -61.8225,B 24.9594,C -1.4727,E1 25.0842,E2 868.0256} C_DIS
LIN {X 67.4891,Y -104.9802,Z 135,A -59.8305,B 24.9596,C -1.4688,E1 25.0888,E2 866.0492} C_DIS
LIN {X 70.7889,Y -102.784,Z 135,A -58.351,B 24.9603,C -1.4551,E1 25.0921,E2 864.607} C_DIS
LIN {X 74.1578,Y -100.3808,Z 135,A -56.4937,B 24.9603,C -1.457,E1 25.0963,E2 862.752} C_DIS
LIN {X 77.4518,Y -97.8617,Z 135,A -54.5701,B 24.9599,C -1.4622,E1 25.1006,E2 860.8232} C_DIS
LIN {X 81.2628,Y -94.7206,Z 135,A -52.2694,B 24.9596,C -1.4691,E1 25.1055,E2 858.515} C_DIS
LIN {X 84.6876,Y -91.6716,Z 135,A -50.233,B 24.9595,C -1.4705,E1 25.1097,E2 856.4834} C_DIS
LIN {X 87.8269,Y -88.6681,Z 135,A -48.5411,B 24.9601,C -1.4599,E1 25.113,E2 854.8237} C_DIS
LIN {X 89.8871,Y -86.5793,Z 135,A -46.7218,B 24.9585,C -1.4876,E1 25.1167,E2 852.9468} C_DIS
LIN {X 93.3951,Y -82.7826,Z 135,A -44.568,B 24.9588,C -1.4824,E1 25.1207,E2 850.8149} C_DIS
LIN {X 95.6324,Y -80.1874,Z 135,A -42.633,B 24.9575,C -1.5053,E1 25.1242,E2 848.8346} C_DIS
LIN {X 98.1323,Y -77.1078,Z 135,A -41.1901,B 24.9584,C -1.4907,E1 25.1267,E2 847.4331} C_DIS
LIN {X 102.0351,Y -71.8639,Z 135,A -38.2217,B 24.958,C -1.4973,E1 25.1316,E2 844.4633} C_DIS
LIN {X 104.4523,Y -68.304,Z 135,A -36.2338,B 24.9576,C -1.5036,E1 25.1346,E2 842.4705} C_DIS
LIN {X 106.6346,Y -64.8439,Z 135,A -34.3609,B 24.9574,C -1.5088,E1 25.1374,E2 840.5948} C_DIS
LIN {X 108.4857,Y -61.6965,Z 135,A -32.6419,B 24.9569,C -1.516,E1 25.1398,E2 838.8678} C_DIS
LIN {X 110.7166,Y -57.5949,Z 135,A -30.5524,B 24.9567,C -1.5196,E1 25.1425,E2 836.7806} C_DIS
LIN {X 112.4955,Y -54.0365,Z 135,A -28.88,B 24.9569,C -1.5172,E1 25.1446,E2 835.1229} C_DIS
LIN {X 113.9641,Y -50.8657,Z 135,A -27.3203,B 24.9567,C -1.5198,E1 25.1464,E2 833.5655} C_DIS
LIN {X 115.0809,Y -48.2862,Z 135,A -25.7581,B 24.9557,C -1.538,E1 25.1481,E2 831.9691} C_DIS
LIN {X 116.8055,Y -43.9506,Z 135,A -23.8578,B 24.956,C -1.5321,E1 25.15,E2 830.0932} C_DIS
LIN {X 118.6917,Y -38.5723,Z 135,A -21.2095,B 24.9554,C -1.5421,E1 25.1524,E2 827.4363} C_DIS
LIN {X 119.7218,Y -35.2403,Z 135,A -19.6596,B 24.9554,C -1.5446,E1 25.1536,E2 825.8894} C_DIS
LIN {X 120.6622,Y -31.8731,Z 135,A -18.084,B 24.9551,C -1.5482,E1 25.1548,E2 824.3142} C_DIS
LIN {X 121.7548,Y -27.4064,Z 135,A -15.8739,B 24.9544,C -1.5602,E1 25.1562,E2 822.0887} C_DIS
LIN {X 122.7249,Y -22.6778,Z 135,A -13.679,B 24.954,C -1.5663,E1 25.1574,E2 819.8923} C_DIS
LIN {X 123.307,Y -19.2514,Z 135,A -12.1907,B 24.954,C -1.566,E1 25.1581,E2 818.4134} C_DIS
LIN {X 123.7922,Y -15.8384,Z 135,A -10.7966,B 24.9543,C -1.5614,E1 25.1586,E2 817.0385} C_DIS
LIN {X 124.1767,Y -12.4765,Z 135,A -8.9692,B 24.9532,C -1.5807,E1 25.1591,E2 815.1762} C_DIS
LIN {X 124.5218,Y -8.3688,Z 135,A -7.1149,B 24.9529,C -1.5849,E1 25.1595,E2 813.323} C_DIS
LIN {X 124.7323,Y -4.1901,Z 135,A -5.1574,B 24.9524,C -1.5932,E1 25.1597,E2 811.3577} C_DIS
LIN {X 124.8037,Y 0.1093,Z 135,A -3.1858,B 24.9521,C -1.5995,E1 25.1597,E2 809.3829} C_DIS
LIN {X 124.737,Y 4.0304,Z 135,A -1.463,B 24.9519,C -1.6014,E1 25.1597,E2 807.6659} C_DIS
LIN {X 124.543,Y 8.0254,Z 135,A 0.3664,B 24.9516,C -1.6071,E1 25.1594,E2 805.8341} C_DIS
LIN {X 124.2298,Y 11.9242,Z 135,A 2.0721,B 24.9516,C -1.6082,E1 25.1589,E2 804.1357} C_DIS
LIN {X 123.7825,Y 15.9125,Z 135,A 3.9224,B 24.9512,C -1.6146,E1 25.1583,E2 802.2813} C_DIS
LIN {X 123.2288,Y 19.7561,Z 135,A 5.7865,B 24.9505,C -1.6245,E1 25.1575,E2 800.4048} C_DIS
LIN {X 122.5603,Y 23.5409,Z 135,A 7.7179,B 24.9497,C -1.6389,E1 25.1565,E2 798.4509} C_DIS
LIN {X 121.4714,Y 28.6401,Z 135,A 9.8768,B 24.95,C -1.6342,E1 25.1552,E2 796.3156} C_DIS
LIN {X 120.5696,Y 32.2201,Z 135,A 11.7443,B 24.9491,C -1.6485,E1 25.1539,E2 794.4252} C_DIS
LIN {X 118.9076,Y 37.8965,Z 135,A 14.1641,B 24.9495,C -1.6415,E1 25.1519,E2 792.0356} C_DIS
LIN {X 117.8527,Y 41.06,Z 135,A 15.7498,B 24.949,C -1.649,E1 25.1505,E2 790.4412} C_DIS
LIN {X 116.4003,Y 45.0128,Z 135,A 17.6429,B 24.9488,C -1.6527,E1 25.1486,E2 788.5498} C_DIS
LIN {X 115.2368,Y 47.9128,Z 135,A 19.0242,B 24.9488,C -1.6542,E1 25.1472,E2 787.1726} C_DIS
LIN {X 113.5864,Y 51.7087,Z 135,A 21.7846,B 24.9456,C -1.7042,E1 25.1439,E2 784.3092} C_DIS
LIN {X 111.0724,Y 56.9046,Z 135,A 23.6928,B 24.9475,C -1.6733,E1 25.1416,E2 782.4841} C_DIS
LIN {X 108.9353,Y 60.8995,Z 135,A 25.7307,B 24.9473,C -1.6769,E1 25.1389,E2 780.4484} C_DIS
LIN {X 106.8898,Y 64.4218,Z 135,A 27.5424,B 24.9472,C -1.679,E1 25.1363,E2 778.641} C_DIS
LIN {X 104.8676,Y 67.6644,Z 135,A 29.3697,B 24.9466,C -1.6874,E1 25.1335,E2 776.8032} C_DIS
LIN {X 102.4883,Y 71.2161,Z 135,A 31.162,B 24.9469,C -1.6838,E1 25.1307,E2 775.0282} C_DIS
LIN {X 100.3217,Y 74.2379,Z 135,A 33.0231,B 24.9461,C -1.696,E1 25.1276,E2 773.1474} C_DIS
LIN {X 98.0052,Y 77.2696,Z 135,A 35.0568,B 24.9449,C -1.7147,E1 25.1241,E2 771.079} C_DIS
LIN {X 95.6396,Y 80.1788,Z 135,A 36.4057,B 24.9459,C -1.6998,E1 25.1217,E2 769.7714} C_DIS
LIN {X 93.5634,Y 82.5922,Z 135,A 37.9982,B 24.9452,C -1.7099,E1 25.1188,E2 768.1623} C_DIS
LIN {X 90.4568,Y 85.9841,Z 135,A 40.0185,B 24.9452,C -1.7099,E1 25.1149,E2 766.1506} C_DIS
LIN {X 87.3654,Y 89.1227,Z 135,A 42.884,B 24.9421,C -1.7573,E1 25.1091,E2 763.1853} C_DIS
LIN {X 82.664,Y 93.4999,Z 135,A 44.7879,B 24.9452,C -1.7102,E1 25.1053,E2 761.4004} C_DIS
LIN {X 80.8996,Y 95.0307,Z 135,A 46.2968,B 24.9436,C -1.7343,E1 25.102,E2 759.8403} C_DIS
LIN {X 78.166,Y 97.2918,Z 135,A 47.5705,B 24.9446,C -1.7195,E1 25.0993,E2 758.6064} C_DIS
LIN {X 74.8699,Y 99.851,Z 135,A 49.5772,B 24.9441,C -1.7276,E1 25.0948,E2 756.5879} C_DIS
LIN {X 71.3403,Y 102.4019,Z 135,A 51.5206,B 24.9441,C -1.7283,E1 25.0904,E2 754.6497} C_DIS
LIN {X 67.7727,Y 104.7974,Z 135,A 53.4873,B 24.9438,C -1.7312,E1 25.0858,E2 752.6826} C_DIS
LIN {X 64.1825,Y 107.0341,Z 135,A 55.4632,B 24.9435,C -1.7359,E1 25.0811,E2 750.7018} C_DIS
LIN {X 60.1182,Y 109.3688,Z 135,A 57.6217,B 24.9433,C -1.7393,E1 25.0759,E2 748.5416} C_DIS
LIN {X 56.6985,Y 111.1773,Z 135,A 59.1897,B 24.9438,C -1.7314,E1 25.072,E2 746.9967} C_DIS
LIN {X 53.9464,Y 112.5386,Z 135,A 60.6568,B 24.9435,C -1.736,E1 25.0683,E2 745.5226} C_DIS
LIN {X 51.1295,Y 113.8461,Z 135,A 62.0247,B 24.9435,C -1.7348,E1 25.0649,E2 744.1609} C_DIS
LIN {X 48.0646,Y 115.1735,Z 135,A 63.7413,B 24.9429,C -1.7455,E1 25.0604,E2 742.423} C_DIS
LIN {X 43.986,Y 116.7922,Z 135,A 65.6385,B 24.9431,C -1.7418,E1 25.0555,E2 740.5389} C_DIS
LIN {X 40.8071,Y 117.9403,Z 135,A 67.1506,B 24.9431,C -1.7412,E1 25.0515,E2 739.0311} C_DIS
LIN {X 38.2675,Y 118.7891,Z 135,A 69.2027,B 24.9404,C -1.7828,E1 25.0458,E2 736.8845} C_DIS
LIN {X 32.8486,Y 120.402,Z 135,A 71.3129,B 24.9419,C -1.7605,E1 25.0403,E2 734.8304} C_DIS
LIN {X 28.5043,Y 121.504,Z 135,A 73.1234,B 24.9426,C -1.7497,E1 25.0355,E2 733.0483} C_DIS
LIN {X 25.2877,Y 122.2125,Z 135,A 74.578,B 24.9428,C -1.7476,E1 25.0315,E2 731.6003} C_DIS
LIN {X 21.9083,Y 122.8626,Z 135,A 76.1674,B 24.9427,C -1.7487,E1 25.0271,E2 730.0101} C_DIS
LIN {X 17.1805,Y 123.6134,Z 135,A 78.3599,B 24.9427,C -1.7491,E1 25.0211,E2 727.8188} C_DIS
LIN {X 13.3734,Y 124.0821,Z 135,A 80.0887,B 24.9427,C -1.7479,E1 25.0163,E2 726.0941} C_DIS
LIN {X 9.4803,Y 124.4408,Z 135,A 81.8838,B 24.9427,C -1.748,E1 25.0113,E2 724.2997} C_DIS
LIN {X 6.1499,Y 124.6492,Z 135,A 83.4278,B 24.9427,C -1.7486,E1 25.007,E2 722.7549} C_DIS
LIN {X 2.5785,Y 124.7752,Z 135,A 85.1303,B 24.9425,C -1.7514,E1 25.0022,E2 721.0462} C_DIS
LIN {X -0.877,Y 124.7979,Z 135,A 86.7416,B 24.9425,C -1.7522,E1 24.9977,E2 719.4328} C_DIS
LIN {X -4.5822,Y 124.717,Z 135,A 88.432,B 24.9425,C -1.7512,E1 24.993,E2 717.7446} C_DIS
LIN {X -9.0346,Y 124.4733,Z 135,A 90.4365,B 24.9427,C -1.7484,E1 24.9874,E2 715.7462} C_DIS
LIN {X -13.0688,Y 124.1149,Z 135,A 92.3607,B 24.9426,C -1.7505,E1 24.9821,E2 713.816} C_DIS
LIN {X -17.3674,Y 123.5867,Z 135,A 94.4775,B 24.9423,C -1.7553,E1 24.9762,E2 711.6861} C_DIS
LIN {X -22.1241,Y 122.824,Z 135,A 97.0597,B 24.9412,C -1.7713,E1 24.969,E2 709.0634} C_DIS
LIN {X -26.5869,Y 121.936,Z 135,A 98.6436,B 24.9429,C -1.7455,E1 24.9648,E2 707.5388} C_DIS
LIN {X -30.3879,Y 121.0448,Z 135,A 100.2094,B 24.9437,C -1.7331,E1 24.9606,E2 706.0003} C_DIS
LIN {X -35.9084,Y 119.5247,Z 135,A 103.0953,B 24.9431,C -1.7423,E1 24.9528,E2 703.088} C_DIS
LIN {X -39.1272,Y 118.5087,Z 135,A 104.5616,B 24.9435,C -1.7366,E1 24.9489,E2 701.6326} C_DIS
LIN {X -44.895,Y 116.4461,Z 135,A 107.4274,B 24.9435,C -1.7353,E1 24.9414,E2 698.7639} C_DIS
LIN {X -48.3558,Y 115.0518,Z 135,A 109.1407,B 24.9437,C -1.7329,E1 24.937,E2 697.0525} C_DIS
LIN {X -52.5286,Y 113.2073,Z 135,A 111.5492,B 24.943,C -1.7443,E1 24.9308,E2 694.611} C_DIS
LIN {X -55.686,Y 111.6891,Z 135,A 112.7943,B 24.9442,C -1.7248,E1 24.9278,E2 693.4091} C_DIS
LIN {X -59.4141,Y 109.7529,Z 135,A 114.8744,B 24.944,C -1.7285,E1 24.9226,E2 691.3144} C_DIS
LIN {X -63.2715,Y 107.5746,Z 135,A 116.8797,B 24.9443,C -1.7235,E1 24.9178,E2 689.315} C_DIS
LIN {X -66.9954,Y 105.2963,Z 135,A 118.9114,B 24.9445,C -1.7209,E1 24.913,E2 687.2829} C_DIS
Enddeposition()
END
